// TIA Portal V20 export
FUNCTION_BLOCK "Sequence_1_JROutPnPLeft"   // FB32846, LAD
TITLE = Sequence
// Sequence template programmend in ladder logic
// stored: IsIECCheckEnabled true, MemoryReserve 100, Namespace Unit1.Em2, SetENOAutomatically true
   VAR_INPUT
      unitStatus : "LAF_typeUnitStatus";
   END_VAR
   VAR
      instSequenceLADControl { ExternalWritable := 'False'} : "LAF_ControlLadSequence";
      instSequenceLADStatus { ExternalWritable := 'False'} : "LAF_StatusLadSequence";
      statTonTime { ExternalWritable := 'False'} : Array[0..9999] of TON_TIME;
      NoDataCheck { S7_SetPoint := 'True'} : "LER_typePartData";
   END_VAR
   VAR_TEMP
      tempCustomerAction : Bool;   // Placeholder for possible actions
      tempDo_nothing_and_wait_for_init : Bool;   // Placeholder for doing nothing
      tempSafeStateCondition : Bool;   // Temp Condition for the equipment module to be in a safe state
   END_VAR
   VAR CONSTANT
      delayTime : Time := T#100ms;
      STEP_IDLE : DInt := 1;
      JOB_1_STEP_01 : DInt := 101;
      JOB_1_STEP_10 : DInt := 110;
      JOB_1_STEP_20 : DInt := 120;
      JOB_1_STEP_30 : DInt := 130;
      JOB_1_STEP_40 : DInt := 140;
      JOB_1_STEP_50 : DInt := 150;
      JOB_1_STEP_60 : DInt := 160;
      JOB_1_STEP_70 : DInt := 170;
      JOB_1_STEP_80 : DInt := 180;
      JOB_1_STEP_90 : DInt := 190;
      JOB_2_STEP_01 : DInt := 201;
      JOB_2_STEP_10 : DInt := 210;
      JOB_2_STEP_11 : DInt := 211;
      JOB_2_STEP_12 : DInt := 212;
      JOB_2_STEP_20 : DInt := 220;
      JOB_2_STEP_21 : DInt := 221;
      JOB_2_STEP_22 : DInt := 222;
      JOB_2_STEP_23 : DInt := 223;
      JOB_2_STEP_30 : DInt := 230;
      JOB_2_STEP_31 : DInt := 231;
      JOB_2_STEP_32 : DInt := 232;
      JOB_2_STEP_33 : DInt := 233;
      JOB_2_STEP_34 : DInt := 234;
      JOB_2_STEP_40 : DInt := 240;
      JOB_2_STEP_41 : DInt := 241;
      JOB_2_STEP_42 : DInt := 242;
      JOB_2_STEP_50 : DInt := 250;
      JOB_2_STEP_60 : DInt := 260;
      JOB_2_STEP_70 : DInt := 270;
      JOB_2_STEP_71 : DInt := 271;
      JOB_2_STEP_72 : DInt := 272;
      JOB_2_STEP_73 : DInt := 273;
      JOB_2_STEP_80 : DInt := 280;
      JOB_2_STEP_90 : DInt := 290;
      JOB_3_STEP_01 : DInt := 301;
      JOB_3_STEP_10 : DInt := 310;
      JOB_3_STEP_11 : DInt := 311;
      JOB_3_STEP_12 : DInt := 312;
      JOB_3_STEP_20 : DInt := 320;
      JOB_3_STEP_21 : DInt := 321;
      JOB_3_STEP_22 : DInt := 322;
      JOB_3_STEP_23 : DInt := 323;
      JOB_3_STEP_30 : DInt := 330;
      JOB_3_STEP_31 : DInt := 331;
      JOB_3_STEP_32 : DInt := 332;
      JOB_3_STEP_33 : DInt := 333;
      JOB_3_STEP_34 : DInt := 334;
      JOB_3_STEP_40 : DInt := 340;
      JOB_3_STEP_41 : DInt := 341;
      JOB_3_STEP_42 : DInt := 342;
      JOB_3_STEP_50 : DInt := 350;
      JOB_3_STEP_60 : DInt := 360;
      JOB_3_STEP_70 : DInt := 370;
      JOB_3_STEP_71 : DInt := 371;
      JOB_3_STEP_72 : DInt := 372;
      JOB_3_STEP_80 : DInt := 380;
      JOB_3_STEP_90 : DInt := 390;
      JOB_4_STEP_01 : DInt := 401;
      JOB_4_STEP_10 : DInt := 410;
      JOB_4_STEP_11 : DInt := 411;
      JOB_4_STEP_12 : DInt := 412;
      JOB_4_STEP_20 : DInt := 420;
      JOB_4_STEP_21 : DInt := 421;
      JOB_4_STEP_22 : DInt := 422;
      JOB_4_STEP_30 : DInt := 430;
      JOB_4_STEP_31 : DInt := 431;
      JOB_4_STEP_32 : DInt := 432;
      JOB_4_STEP_40 : DInt := 440;
      JOB_4_STEP_41 : DInt := 441;
      JOB_4_STEP_42 : DInt := 442;
      JOB_4_STEP_50 : DInt := 450;
      JOB_4_STEP_51 : DInt := 451;
      JOB_4_STEP_52 : DInt := 452;
      JOB_4_STEP_60 : DInt := 460;
      JOB_4_STEP_70 : DInt := 470;
      JOB_4_STEP_80 : DInt := 480;
      JOB_4_STEP_90 : DInt := 490;
      STEP_IMMEDIATE_STOP : DInt := 9001;   // Step executed when an immediate stop command is triggered for the sequence (i.e. when unit is in state aborting)
      TRUE : Bool := TRUE;
      FALSE : Bool := FALSE;
   END_VAR
   VAR_TEMP   // added for the SCL form of the ladder/FBD networks
      _w1 : Bool;
      _w2 : Bool;
      _w3 : Bool;
      _w4 : Bool;
      _w5 : Bool;
      _w6 : Bool;
      _w7 : Bool;
   END_VAR
BEGIN

REGION Network 1: BLOCK INFO HEADER
   // (company) / (C) Copyright (year)
   // ---------------------------------------------------------------------------------
   // Title:                             (Title of this block)
   // Comment/Function: (that is implemented in the block)
   // Library/Family:           (that the source is dedicated to)
   // Author:                        (department / person in charge / contact)
   // Target System:          (test system with FW version)
   // Engineering:              TIA Portal (SW version)
   // Restrictions:               (OB types, etc.)
   // Requirements:           (hardware, technological package, etc.)
   // ---------------------------------------------------------------------------------
   // Change log table:
   // Version          | Date             | Signature      | Expert in charge  | Changes applied ------------------------|----------------------|-------------------------|--------------------------------|-----------------------
   // 001.000.000 | yyyy-mm-dd | 0x00000000 | (name of expert) | First released version
END_REGION

REGION Network 2: DESCRIPTION
   // This is a template block provided by the Automation Framework. It can be used to create an own project.
   // The Block Info Header is prepared to put in your own data.
   // Description of the block could be added here and the docu created by Code2Docu.
END_REGION

REGION Network 3: *************** CONTROL **********************
END_REGION

REGION Network 4: Sequence Control ("Enter your Sequins number here")
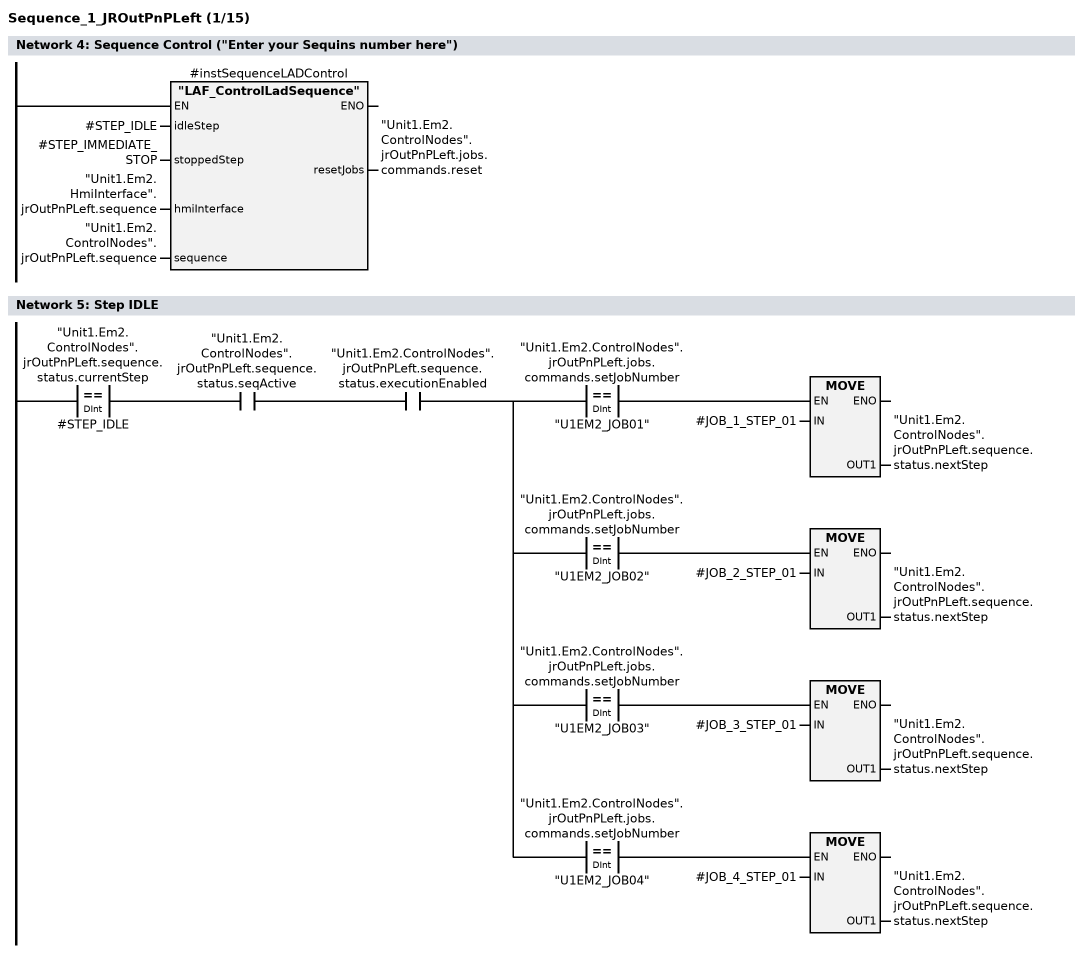
   RUNG wire#powerrail
      #instSequenceLADControl(idleStep := #STEP_IDLE, stoppedStep := #STEP_IMMEDIATE_STOP, hmiInterface := "Unit1.Em2.HmiInterface".jrOutPnPLeft.sequence, sequence := "Unit1.Em2.ControlNodes".jrOutPnPLeft.sequence, resetJobs => "Unit1.Em2.ControlNodes".jrOutPnPLeft.jobs.commands.reset)
   END_RUNG
   // the same network as SCL:
   #instSequenceLADControl(idleStep := #STEP_IDLE,   // "LAF_ControlLadSequence"
                           stoppedStep := #STEP_IMMEDIATE_STOP,
                           hmiInterface := "Unit1.Em2.HmiInterface".jrOutPnPLeft.sequence,
                           sequence := "Unit1.Em2.ControlNodes".jrOutPnPLeft.sequence,
                           resetJobs => "Unit1.Em2.ControlNodes".jrOutPnPLeft.jobs.commands.reset);
END_REGION

REGION Network 5: Step IDLE
   RUNG wire#powerrail
      { S7_Templates := "SrcType := DInt" } EQ_Contact(in1 := "Unit1.Em2.ControlNodes".jrOutPnPLeft.sequence.status.currentStep, in2 := #STEP_IDLE)
      Contact( "Unit1.Em2.ControlNodes".jrOutPnPLeft.sequence.status.seqActive )
      Contact( "Unit1.Em2.ControlNodes".jrOutPnPLeft.sequence.status.executionEnabled )
      wire#w1
      { S7_Templates := "SrcType := DInt" } EQ_Contact(in1 := "Unit1.Em2.ControlNodes".jrOutPnPLeft.jobs.commands.setJobNumber, in2 := "U1EM2_JOB01")
      Move(in := #JOB_1_STEP_01, out1 => "Unit1.Em2.ControlNodes".jrOutPnPLeft.sequence.status.nextStep)
   END_RUNG
   RUNG wire#w1
      { S7_Templates := "SrcType := DInt" } EQ_Contact(in1 := "Unit1.Em2.ControlNodes".jrOutPnPLeft.jobs.commands.setJobNumber, in2 := "U1EM2_JOB02")
      Move(in := #JOB_2_STEP_01, out1 => "Unit1.Em2.ControlNodes".jrOutPnPLeft.sequence.status.nextStep)
   END_RUNG
   RUNG wire#w1
      { S7_Templates := "SrcType := DInt" } EQ_Contact(in1 := "Unit1.Em2.ControlNodes".jrOutPnPLeft.jobs.commands.setJobNumber, in2 := "U1EM2_JOB03")
      Move(in := #JOB_3_STEP_01, out1 => "Unit1.Em2.ControlNodes".jrOutPnPLeft.sequence.status.nextStep)
   END_RUNG
   RUNG wire#w1
      { S7_Templates := "SrcType := DInt" } EQ_Contact(in1 := "Unit1.Em2.ControlNodes".jrOutPnPLeft.jobs.commands.setJobNumber, in2 := "U1EM2_JOB04")
      Move(in := #JOB_4_STEP_01, out1 => "Unit1.Em2.ControlNodes".jrOutPnPLeft.sequence.status.nextStep)
   END_RUNG
   // the same network as SCL:
   #_w1 := ("Unit1.Em2.ControlNodes".jrOutPnPLeft.sequence.status.currentStep = #STEP_IDLE) AND "Unit1.Em2.ControlNodes".jrOutPnPLeft.sequence.status.seqActive AND "Unit1.Em2.ControlNodes".jrOutPnPLeft.sequence.status.executionEnabled;
   IF #_w1 AND ("Unit1.Em2.ControlNodes".jrOutPnPLeft.jobs.commands.setJobNumber = "U1EM2_JOB01") THEN
       "Unit1.Em2.ControlNodes".jrOutPnPLeft.sequence.status.nextStep := #JOB_1_STEP_01;
   END_IF;
   IF #_w1 AND ("Unit1.Em2.ControlNodes".jrOutPnPLeft.jobs.commands.setJobNumber = "U1EM2_JOB02") THEN
       "Unit1.Em2.ControlNodes".jrOutPnPLeft.sequence.status.nextStep := #JOB_2_STEP_01;
   END_IF;
   IF #_w1 AND ("Unit1.Em2.ControlNodes".jrOutPnPLeft.jobs.commands.setJobNumber = "U1EM2_JOB03") THEN
       "Unit1.Em2.ControlNodes".jrOutPnPLeft.sequence.status.nextStep := #JOB_3_STEP_01;
   END_IF;
   IF #_w1 AND ("Unit1.Em2.ControlNodes".jrOutPnPLeft.jobs.commands.setJobNumber = "U1EM2_JOB04") THEN
       "Unit1.Em2.ControlNodes".jrOutPnPLeft.sequence.status.nextStep := #JOB_4_STEP_01;
   END_IF;
END_REGION

REGION Network 6: *************** JOB[1] EM HOMING *************************
END_REGION

REGION Network 7: Step[101] : JOB[1] Condition
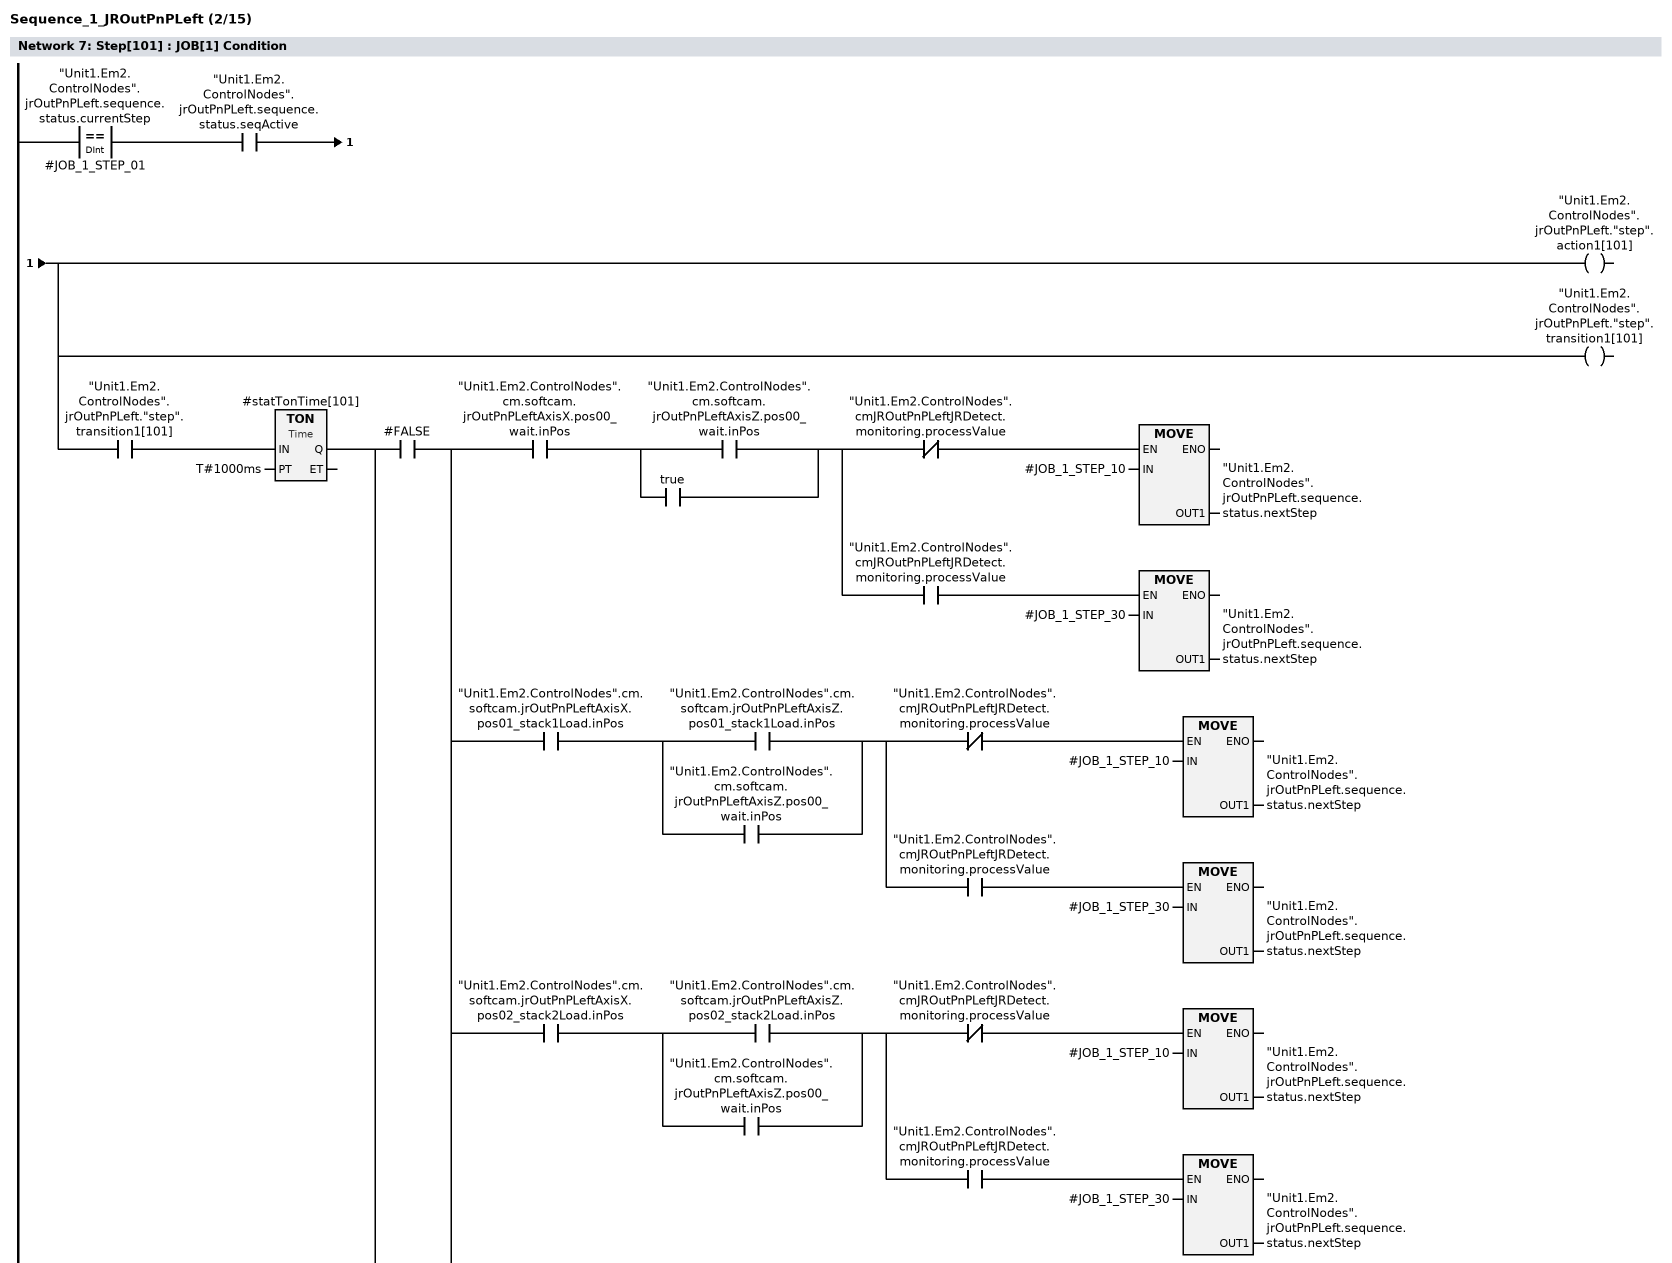
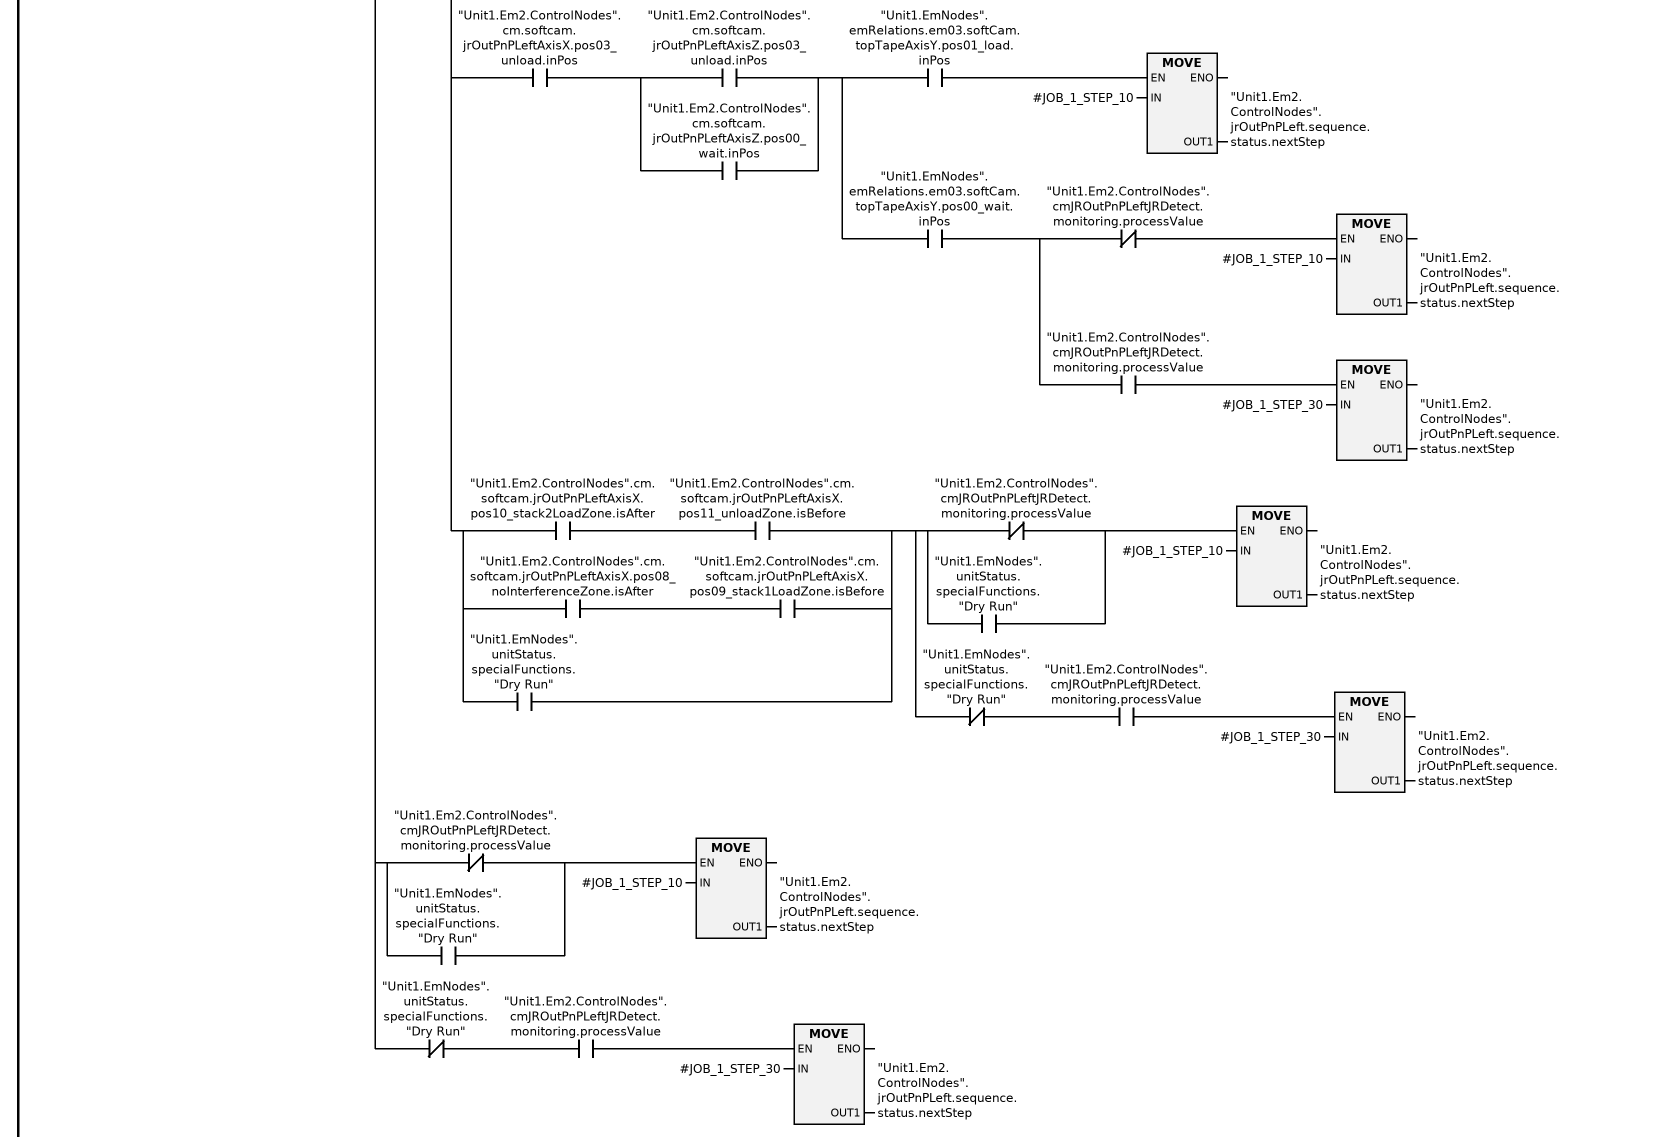
   RUNG wire#powerrail
      { S7_Templates := "SrcType := DInt" } EQ_Contact(in1 := "Unit1.Em2.ControlNodes".jrOutPnPLeft.sequence.status.currentStep, in2 := #JOB_1_STEP_01)
      Contact( "Unit1.Em2.ControlNodes".jrOutPnPLeft.sequence.status.seqActive )
      wire#w1
      Coil( "Unit1.Em2.ControlNodes".jrOutPnPLeft."step".action1[101] )
   END_RUNG
   RUNG wire#w1
      Coil( "Unit1.Em2.ControlNodes".jrOutPnPLeft."step".transition1[101] )
   END_RUNG
   RUNG wire#w1
      Contact( "Unit1.Em2.ControlNodes".jrOutPnPLeft."step".transition1[101] )
      { S7_Templates := "time_type := Time" } #statTonTime[101].TON(pt := T#1000ms, et =>)
      wire#w2
      Contact( #FALSE )
      wire#w3
      Contact( "Unit1.Em2.ControlNodes".cm.softcam.jrOutPnPLeftAxisX.pos00_wait.inPos )
      wire#w4
      Contact( "Unit1.Em2.ControlNodes".cm.softcam.jrOutPnPLeftAxisZ.pos00_wait.inPos )
      wire#w5
      I_Contact( "Unit1.Em2.ControlNodes".cmJROutPnPLeftJRDetect.monitoring.processValue )
      Move(in := #JOB_1_STEP_10, out1 => "Unit1.Em2.ControlNodes".jrOutPnPLeft.sequence.status.nextStep)
   END_RUNG
   RUNG wire#w4
      Contact( true )
   END_RUNG wire#w5
   RUNG wire#w5
      Contact( "Unit1.Em2.ControlNodes".cmJROutPnPLeftJRDetect.monitoring.processValue )
      Move(in := #JOB_1_STEP_30, out1 => "Unit1.Em2.ControlNodes".jrOutPnPLeft.sequence.status.nextStep)
   END_RUNG
   RUNG wire#w3
      Contact( "Unit1.Em2.ControlNodes".cm.softcam.jrOutPnPLeftAxisX.pos01_stack1Load.inPos )
      wire#w6
      Contact( "Unit1.Em2.ControlNodes".cm.softcam.jrOutPnPLeftAxisZ.pos01_stack1Load.inPos )
      wire#w7
      I_Contact( "Unit1.Em2.ControlNodes".cmJROutPnPLeftJRDetect.monitoring.processValue )
      Move(in := #JOB_1_STEP_10, out1 => "Unit1.Em2.ControlNodes".jrOutPnPLeft.sequence.status.nextStep)
   END_RUNG
   RUNG wire#w6
      Contact( "Unit1.Em2.ControlNodes".cm.softcam.jrOutPnPLeftAxisZ.pos00_wait.inPos )
   END_RUNG wire#w7
   RUNG wire#w7
      Contact( "Unit1.Em2.ControlNodes".cmJROutPnPLeftJRDetect.monitoring.processValue )
      Move(in := #JOB_1_STEP_30, out1 => "Unit1.Em2.ControlNodes".jrOutPnPLeft.sequence.status.nextStep)
   END_RUNG
   RUNG wire#w3
      Contact( "Unit1.Em2.ControlNodes".cm.softcam.jrOutPnPLeftAxisX.pos02_stack2Load.inPos )
      wire#w8
      Contact( "Unit1.Em2.ControlNodes".cm.softcam.jrOutPnPLeftAxisZ.pos02_stack2Load.inPos )
      wire#w9
      I_Contact( "Unit1.Em2.ControlNodes".cmJROutPnPLeftJRDetect.monitoring.processValue )
      Move(in := #JOB_1_STEP_10, out1 => "Unit1.Em2.ControlNodes".jrOutPnPLeft.sequence.status.nextStep)
   END_RUNG
   RUNG wire#w8
      Contact( "Unit1.Em2.ControlNodes".cm.softcam.jrOutPnPLeftAxisZ.pos00_wait.inPos )
   END_RUNG wire#w9
   RUNG wire#w9
      Contact( "Unit1.Em2.ControlNodes".cmJROutPnPLeftJRDetect.monitoring.processValue )
      Move(in := #JOB_1_STEP_30, out1 => "Unit1.Em2.ControlNodes".jrOutPnPLeft.sequence.status.nextStep)
   END_RUNG
   RUNG wire#w3
      Contact( "Unit1.Em2.ControlNodes".cm.softcam.jrOutPnPLeftAxisX.pos03_unload.inPos )
      wire#w10
      Contact( "Unit1.Em2.ControlNodes".cm.softcam.jrOutPnPLeftAxisZ.pos03_unload.inPos )
      wire#w11
      Contact( "Unit1.EmNodes".emRelations.em03.softCam.topTapeAxisY.pos01_load.inPos )
      Move(in := #JOB_1_STEP_10, out1 => "Unit1.Em2.ControlNodes".jrOutPnPLeft.sequence.status.nextStep)
   END_RUNG
   RUNG wire#w10
      Contact( "Unit1.Em2.ControlNodes".cm.softcam.jrOutPnPLeftAxisZ.pos00_wait.inPos )
   END_RUNG wire#w11
   RUNG wire#w11
      Contact( "Unit1.EmNodes".emRelations.em03.softCam.topTapeAxisY.pos00_wait.inPos )
      wire#w12
      I_Contact( "Unit1.Em2.ControlNodes".cmJROutPnPLeftJRDetect.monitoring.processValue )
      Move(in := #JOB_1_STEP_10, out1 => "Unit1.Em2.ControlNodes".jrOutPnPLeft.sequence.status.nextStep)
   END_RUNG
   RUNG wire#w12
      Contact( "Unit1.Em2.ControlNodes".cmJROutPnPLeftJRDetect.monitoring.processValue )
      Move(in := #JOB_1_STEP_30, out1 => "Unit1.Em2.ControlNodes".jrOutPnPLeft.sequence.status.nextStep)
   END_RUNG
   RUNG wire#w3
      Contact( "Unit1.Em2.ControlNodes".cm.softcam.jrOutPnPLeftAxisX.pos10_stack2LoadZone.isAfter )
      Contact( "Unit1.Em2.ControlNodes".cm.softcam.jrOutPnPLeftAxisX.pos11_unloadZone.isBefore )
      wire#w13
      I_Contact( "Unit1.Em2.ControlNodes".cmJROutPnPLeftJRDetect.monitoring.processValue )
      wire#w14
      Move(in := #JOB_1_STEP_10, out1 => "Unit1.Em2.ControlNodes".jrOutPnPLeft.sequence.status.nextStep)
   END_RUNG
   RUNG wire#w3
      Contact( "Unit1.Em2.ControlNodes".cm.softcam.jrOutPnPLeftAxisX.pos08_noInterferenceZone.isAfter )
      Contact( "Unit1.Em2.ControlNodes".cm.softcam.jrOutPnPLeftAxisX.pos09_stack1LoadZone.isBefore )
   END_RUNG wire#w13
   RUNG wire#w3
      Contact( "Unit1.EmNodes".unitStatus.specialFunctions."Dry Run" )
   END_RUNG wire#w13
   RUNG wire#w13
      Contact( "Unit1.EmNodes".unitStatus.specialFunctions."Dry Run" )
   END_RUNG wire#w14
   RUNG wire#w13
      I_Contact( "Unit1.EmNodes".unitStatus.specialFunctions."Dry Run" )
      Contact( "Unit1.Em2.ControlNodes".cmJROutPnPLeftJRDetect.monitoring.processValue )
      Move(in := #JOB_1_STEP_30, out1 => "Unit1.Em2.ControlNodes".jrOutPnPLeft.sequence.status.nextStep)
   END_RUNG
   RUNG wire#w2
      I_Contact( "Unit1.Em2.ControlNodes".cmJROutPnPLeftJRDetect.monitoring.processValue )
      wire#w15
      Move(in := #JOB_1_STEP_10, out1 => "Unit1.Em2.ControlNodes".jrOutPnPLeft.sequence.status.nextStep)
   END_RUNG
   RUNG wire#w2
      Contact( "Unit1.EmNodes".unitStatus.specialFunctions."Dry Run" )
   END_RUNG wire#w15
   RUNG wire#w2
      I_Contact( "Unit1.EmNodes".unitStatus.specialFunctions."Dry Run" )
      Contact( "Unit1.Em2.ControlNodes".cmJROutPnPLeftJRDetect.monitoring.processValue )
      Move(in := #JOB_1_STEP_30, out1 => "Unit1.Em2.ControlNodes".jrOutPnPLeft.sequence.status.nextStep)
   END_RUNG
   // the same network as SCL:
   "Unit1.Em2.ControlNodes".jrOutPnPLeft."step".action1[101] := ("Unit1.Em2.ControlNodes".jrOutPnPLeft.sequence.status.currentStep = #JOB_1_STEP_01) AND "Unit1.Em2.ControlNodes".jrOutPnPLeft.sequence.status.seqActive;
   "Unit1.Em2.ControlNodes".jrOutPnPLeft."step".transition1[101] := ("Unit1.Em2.ControlNodes".jrOutPnPLeft.sequence.status.currentStep = #JOB_1_STEP_01) AND "Unit1.Em2.ControlNodes".jrOutPnPLeft.sequence.status.seqActive;
   #statTonTime[101].TON(IN := ("Unit1.Em2.ControlNodes".jrOutPnPLeft.sequence.status.currentStep = #JOB_1_STEP_01) AND "Unit1.Em2.ControlNodes".jrOutPnPLeft.sequence.status.seqActive AND "Unit1.Em2.ControlNodes".jrOutPnPLeft."step".transition1[101],
                         PT := T#1000ms);
   #_w1 := #statTonTime[101].Q AND #FALSE;
   #_w2 := #_w1 AND "Unit1.Em2.ControlNodes".cm.softcam.jrOutPnPLeftAxisX.pos00_wait.inPos AND ("Unit1.Em2.ControlNodes".cm.softcam.jrOutPnPLeftAxisZ.pos00_wait.inPos OR true);
   IF #_w2 AND NOT "Unit1.Em2.ControlNodes".cmJROutPnPLeftJRDetect.monitoring.processValue THEN
       "Unit1.Em2.ControlNodes".jrOutPnPLeft.sequence.status.nextStep := #JOB_1_STEP_10;
   END_IF;
   IF #_w2 AND "Unit1.Em2.ControlNodes".cmJROutPnPLeftJRDetect.monitoring.processValue THEN
       "Unit1.Em2.ControlNodes".jrOutPnPLeft.sequence.status.nextStep := #JOB_1_STEP_30;
   END_IF;
   #_w3 := #_w1 AND "Unit1.Em2.ControlNodes".cm.softcam.jrOutPnPLeftAxisX.pos01_stack1Load.inPos AND ("Unit1.Em2.ControlNodes".cm.softcam.jrOutPnPLeftAxisZ.pos01_stack1Load.inPos OR "Unit1.Em2.ControlNodes".cm.softcam.jrOutPnPLeftAxisZ.pos00_wait.inPos);
   IF #_w3 AND NOT "Unit1.Em2.ControlNodes".cmJROutPnPLeftJRDetect.monitoring.processValue THEN
       "Unit1.Em2.ControlNodes".jrOutPnPLeft.sequence.status.nextStep := #JOB_1_STEP_10;
   END_IF;
   IF #_w3 AND "Unit1.Em2.ControlNodes".cmJROutPnPLeftJRDetect.monitoring.processValue THEN
       "Unit1.Em2.ControlNodes".jrOutPnPLeft.sequence.status.nextStep := #JOB_1_STEP_30;
   END_IF;
   #_w4 := #_w1 AND "Unit1.Em2.ControlNodes".cm.softcam.jrOutPnPLeftAxisX.pos02_stack2Load.inPos AND ("Unit1.Em2.ControlNodes".cm.softcam.jrOutPnPLeftAxisZ.pos02_stack2Load.inPos OR "Unit1.Em2.ControlNodes".cm.softcam.jrOutPnPLeftAxisZ.pos00_wait.inPos);
   IF #_w4 AND NOT "Unit1.Em2.ControlNodes".cmJROutPnPLeftJRDetect.monitoring.processValue THEN
       "Unit1.Em2.ControlNodes".jrOutPnPLeft.sequence.status.nextStep := #JOB_1_STEP_10;
   END_IF;
   IF #_w4 AND "Unit1.Em2.ControlNodes".cmJROutPnPLeftJRDetect.monitoring.processValue THEN
       "Unit1.Em2.ControlNodes".jrOutPnPLeft.sequence.status.nextStep := #JOB_1_STEP_30;
   END_IF;
   #_w5 := #_w1 AND "Unit1.Em2.ControlNodes".cm.softcam.jrOutPnPLeftAxisX.pos03_unload.inPos AND ("Unit1.Em2.ControlNodes".cm.softcam.jrOutPnPLeftAxisZ.pos03_unload.inPos OR "Unit1.Em2.ControlNodes".cm.softcam.jrOutPnPLeftAxisZ.pos00_wait.inPos);
   IF #_w5 AND "Unit1.EmNodes".emRelations.em03.softCam.topTapeAxisY.pos01_load.inPos THEN
       "Unit1.Em2.ControlNodes".jrOutPnPLeft.sequence.status.nextStep := #JOB_1_STEP_10;
   END_IF;
   #_w6 := #_w5 AND "Unit1.EmNodes".emRelations.em03.softCam.topTapeAxisY.pos00_wait.inPos;
   IF #_w6 AND NOT "Unit1.Em2.ControlNodes".cmJROutPnPLeftJRDetect.monitoring.processValue THEN
       "Unit1.Em2.ControlNodes".jrOutPnPLeft.sequence.status.nextStep := #JOB_1_STEP_10;
   END_IF;
   IF #_w6 AND "Unit1.Em2.ControlNodes".cmJROutPnPLeftJRDetect.monitoring.processValue THEN
       "Unit1.Em2.ControlNodes".jrOutPnPLeft.sequence.status.nextStep := #JOB_1_STEP_30;
   END_IF;
   #_w7 := #_w1 AND (("Unit1.Em2.ControlNodes".cm.softcam.jrOutPnPLeftAxisX.pos10_stack2LoadZone.isAfter AND "Unit1.Em2.ControlNodes".cm.softcam.jrOutPnPLeftAxisX.pos11_unloadZone.isBefore) OR ("Unit1.Em2.ControlNodes".cm.softcam.jrOutPnPLeftAxisX.pos08_noInterferenceZone.isAfter AND "Unit1.Em2.ControlNodes".cm.softcam.jrOutPnPLeftAxisX.pos09_stack1LoadZone.isBefore) OR "Unit1.EmNodes".unitStatus.specialFunctions."Dry Run");
   IF #_w7 AND (NOT "Unit1.Em2.ControlNodes".cmJROutPnPLeftJRDetect.monitoring.processValue OR "Unit1.EmNodes".unitStatus.specialFunctions."Dry Run") THEN
       "Unit1.Em2.ControlNodes".jrOutPnPLeft.sequence.status.nextStep := #JOB_1_STEP_10;
   END_IF;
   IF #_w7 AND NOT "Unit1.EmNodes".unitStatus.specialFunctions."Dry Run" AND "Unit1.Em2.ControlNodes".cmJROutPnPLeftJRDetect.monitoring.processValue THEN
       "Unit1.Em2.ControlNodes".jrOutPnPLeft.sequence.status.nextStep := #JOB_1_STEP_30;
   END_IF;
   IF #statTonTime[101].Q AND (NOT "Unit1.Em2.ControlNodes".cmJROutPnPLeftJRDetect.monitoring.processValue OR "Unit1.EmNodes".unitStatus.specialFunctions."Dry Run") THEN
       "Unit1.Em2.ControlNodes".jrOutPnPLeft.sequence.status.nextStep := #JOB_1_STEP_10;
   END_IF;
   IF #statTonTime[101].Q AND NOT "Unit1.EmNodes".unitStatus.specialFunctions."Dry Run" AND "Unit1.Em2.ControlNodes".cmJROutPnPLeftJRDetect.monitoring.processValue THEN
       "Unit1.Em2.ControlNodes".jrOutPnPLeft.sequence.status.nextStep := #JOB_1_STEP_30;
   END_IF;
END_REGION

REGION Network 8: Step[110] : JR PP Left Clamp Open
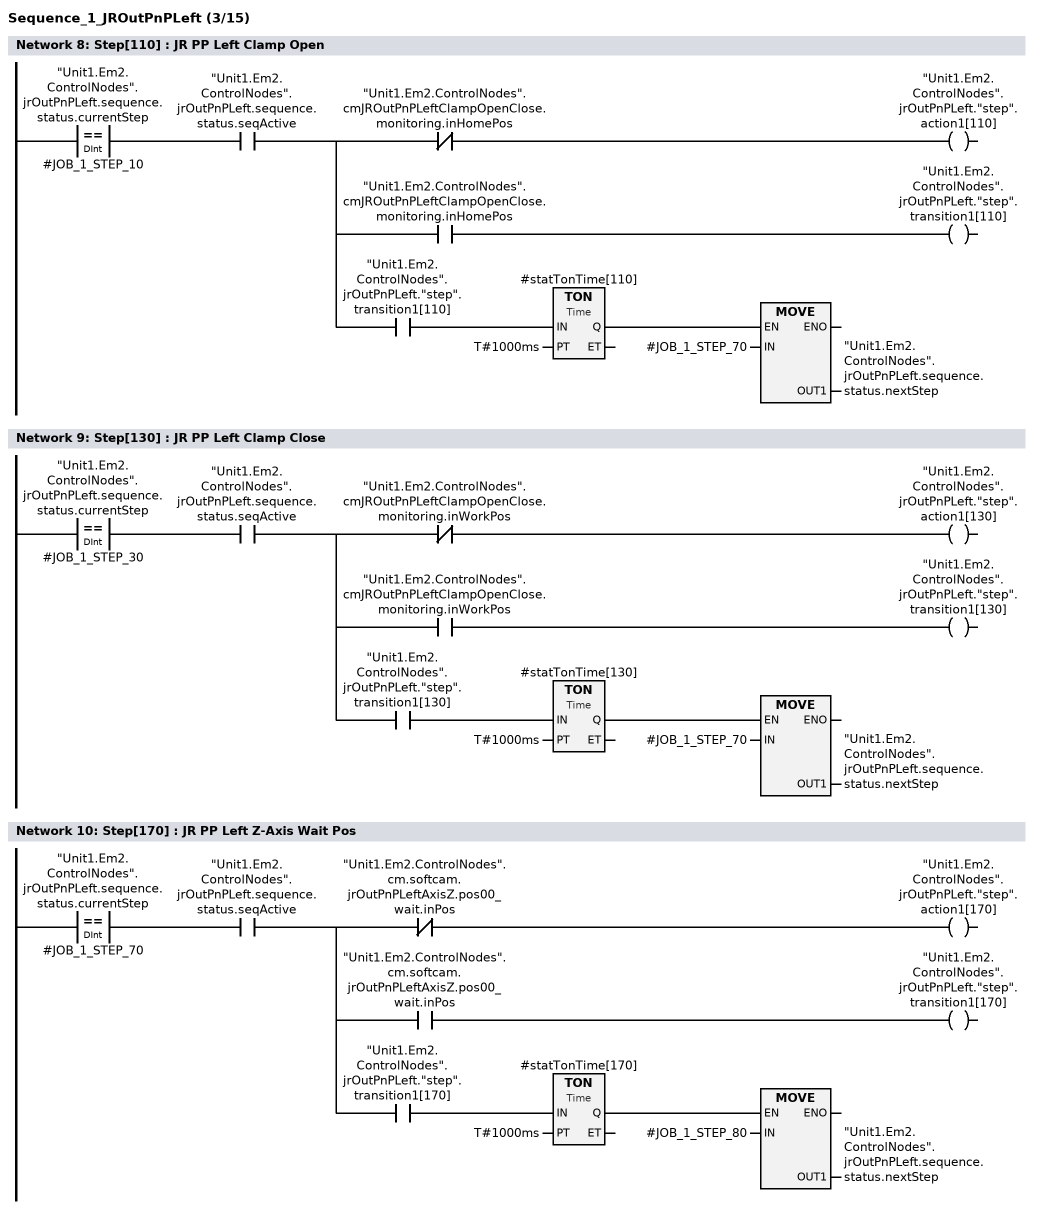
   RUNG wire#powerrail
      { S7_Templates := "SrcType := DInt" } EQ_Contact(in1 := "Unit1.Em2.ControlNodes".jrOutPnPLeft.sequence.status.currentStep, in2 := #JOB_1_STEP_10)
      Contact( "Unit1.Em2.ControlNodes".jrOutPnPLeft.sequence.status.seqActive )
      wire#w1
      I_Contact( "Unit1.Em2.ControlNodes".cmJROutPnPLeftClampOpenClose.monitoring.inHomePos )
      Coil( "Unit1.Em2.ControlNodes".jrOutPnPLeft."step".action1[110] )
   END_RUNG
   RUNG wire#w1
      Contact( "Unit1.Em2.ControlNodes".cmJROutPnPLeftClampOpenClose.monitoring.inHomePos )
      Coil( "Unit1.Em2.ControlNodes".jrOutPnPLeft."step".transition1[110] )
   END_RUNG
   RUNG wire#w1
      Contact( "Unit1.Em2.ControlNodes".jrOutPnPLeft."step".transition1[110] )
      { S7_Templates := "time_type := Time" } #statTonTime[110].TON(pt := T#1000ms, et =>)
      Move(in := #JOB_1_STEP_70, out1 => "Unit1.Em2.ControlNodes".jrOutPnPLeft.sequence.status.nextStep)
   END_RUNG
   // the same network as SCL:
   #_w1 := ("Unit1.Em2.ControlNodes".jrOutPnPLeft.sequence.status.currentStep = #JOB_1_STEP_10) AND "Unit1.Em2.ControlNodes".jrOutPnPLeft.sequence.status.seqActive;
   "Unit1.Em2.ControlNodes".jrOutPnPLeft."step".action1[110] := #_w1 AND NOT "Unit1.Em2.ControlNodes".cmJROutPnPLeftClampOpenClose.monitoring.inHomePos;
   "Unit1.Em2.ControlNodes".jrOutPnPLeft."step".transition1[110] := #_w1 AND "Unit1.Em2.ControlNodes".cmJROutPnPLeftClampOpenClose.monitoring.inHomePos;
   #statTonTime[110].TON(IN := #_w1 AND "Unit1.Em2.ControlNodes".jrOutPnPLeft."step".transition1[110],
                         PT := T#1000ms);
   IF #statTonTime[110].Q THEN
       "Unit1.Em2.ControlNodes".jrOutPnPLeft.sequence.status.nextStep := #JOB_1_STEP_70;
   END_IF;
END_REGION

REGION Network 9: Step[130] : JR PP Left Clamp Close
   RUNG wire#powerrail
      { S7_Templates := "SrcType := DInt" } EQ_Contact(in1 := "Unit1.Em2.ControlNodes".jrOutPnPLeft.sequence.status.currentStep, in2 := #JOB_1_STEP_30)
      Contact( "Unit1.Em2.ControlNodes".jrOutPnPLeft.sequence.status.seqActive )
      wire#w1
      I_Contact( "Unit1.Em2.ControlNodes".cmJROutPnPLeftClampOpenClose.monitoring.inWorkPos )
      Coil( "Unit1.Em2.ControlNodes".jrOutPnPLeft."step".action1[130] )
   END_RUNG
   RUNG wire#w1
      Contact( "Unit1.Em2.ControlNodes".cmJROutPnPLeftClampOpenClose.monitoring.inWorkPos )
      Coil( "Unit1.Em2.ControlNodes".jrOutPnPLeft."step".transition1[130] )
   END_RUNG
   RUNG wire#w1
      Contact( "Unit1.Em2.ControlNodes".jrOutPnPLeft."step".transition1[130] )
      { S7_Templates := "time_type := Time" } #statTonTime[130].TON(pt := T#1000ms, et =>)
      Move(in := #JOB_1_STEP_70, out1 => "Unit1.Em2.ControlNodes".jrOutPnPLeft.sequence.status.nextStep)
   END_RUNG
   // the same network as SCL:
   #_w1 := ("Unit1.Em2.ControlNodes".jrOutPnPLeft.sequence.status.currentStep = #JOB_1_STEP_30) AND "Unit1.Em2.ControlNodes".jrOutPnPLeft.sequence.status.seqActive;
   "Unit1.Em2.ControlNodes".jrOutPnPLeft."step".action1[130] := #_w1 AND NOT "Unit1.Em2.ControlNodes".cmJROutPnPLeftClampOpenClose.monitoring.inWorkPos;
   "Unit1.Em2.ControlNodes".jrOutPnPLeft."step".transition1[130] := #_w1 AND "Unit1.Em2.ControlNodes".cmJROutPnPLeftClampOpenClose.monitoring.inWorkPos;
   #statTonTime[130].TON(IN := #_w1 AND "Unit1.Em2.ControlNodes".jrOutPnPLeft."step".transition1[130],
                         PT := T#1000ms);
   IF #statTonTime[130].Q THEN
       "Unit1.Em2.ControlNodes".jrOutPnPLeft.sequence.status.nextStep := #JOB_1_STEP_70;
   END_IF;
END_REGION

REGION Network 10: Step[170] : JR PP Left Z-Axis Wait Pos
   RUNG wire#powerrail
      { S7_Templates := "SrcType := DInt" } EQ_Contact(in1 := "Unit1.Em2.ControlNodes".jrOutPnPLeft.sequence.status.currentStep, in2 := #JOB_1_STEP_70)
      Contact( "Unit1.Em2.ControlNodes".jrOutPnPLeft.sequence.status.seqActive )
      wire#w1
      I_Contact( "Unit1.Em2.ControlNodes".cm.softcam.jrOutPnPLeftAxisZ.pos00_wait.inPos )
      Coil( "Unit1.Em2.ControlNodes".jrOutPnPLeft."step".action1[170] )
   END_RUNG
   RUNG wire#w1
      Contact( "Unit1.Em2.ControlNodes".cm.softcam.jrOutPnPLeftAxisZ.pos00_wait.inPos )
      Coil( "Unit1.Em2.ControlNodes".jrOutPnPLeft."step".transition1[170] )
   END_RUNG
   RUNG wire#w1
      Contact( "Unit1.Em2.ControlNodes".jrOutPnPLeft."step".transition1[170] )
      { S7_Templates := "time_type := Time" } #statTonTime[170].TON(pt := T#1000ms, et =>)
      Move(in := #JOB_1_STEP_80, out1 => "Unit1.Em2.ControlNodes".jrOutPnPLeft.sequence.status.nextStep)
   END_RUNG
   // the same network as SCL:
   #_w1 := ("Unit1.Em2.ControlNodes".jrOutPnPLeft.sequence.status.currentStep = #JOB_1_STEP_70) AND "Unit1.Em2.ControlNodes".jrOutPnPLeft.sequence.status.seqActive;
   "Unit1.Em2.ControlNodes".jrOutPnPLeft."step".action1[170] := #_w1 AND NOT "Unit1.Em2.ControlNodes".cm.softcam.jrOutPnPLeftAxisZ.pos00_wait.inPos;
   "Unit1.Em2.ControlNodes".jrOutPnPLeft."step".transition1[170] := #_w1 AND "Unit1.Em2.ControlNodes".cm.softcam.jrOutPnPLeftAxisZ.pos00_wait.inPos;
   #statTonTime[170].TON(IN := #_w1 AND "Unit1.Em2.ControlNodes".jrOutPnPLeft."step".transition1[170],
                         PT := T#1000ms);
   IF #statTonTime[170].Q THEN
       "Unit1.Em2.ControlNodes".jrOutPnPLeft.sequence.status.nextStep := #JOB_1_STEP_80;
   END_IF;
END_REGION

REGION Network 11: Step[180] : JR PP Left X-Axis Wait Pos
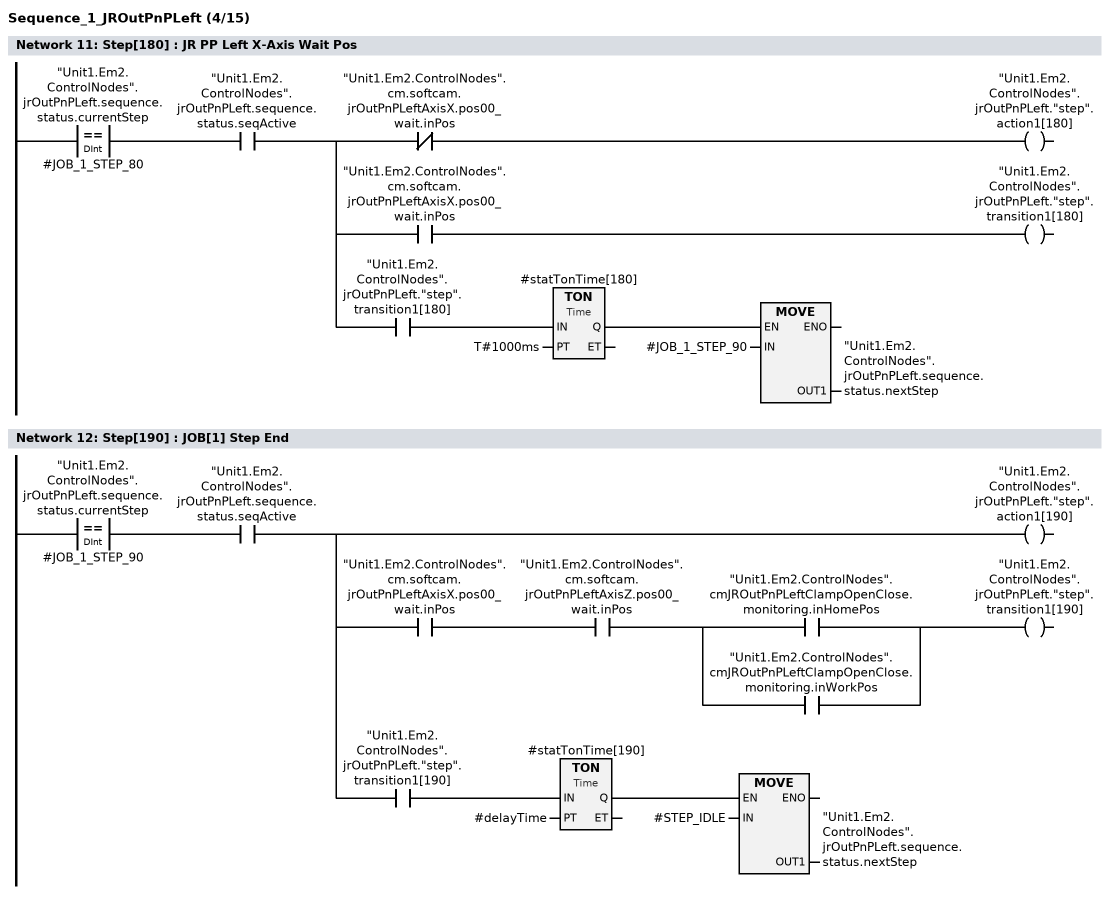
   RUNG wire#powerrail
      { S7_Templates := "SrcType := DInt" } EQ_Contact(in1 := "Unit1.Em2.ControlNodes".jrOutPnPLeft.sequence.status.currentStep, in2 := #JOB_1_STEP_80)
      Contact( "Unit1.Em2.ControlNodes".jrOutPnPLeft.sequence.status.seqActive )
      wire#w1
      I_Contact( "Unit1.Em2.ControlNodes".cm.softcam.jrOutPnPLeftAxisX.pos00_wait.inPos )
      Coil( "Unit1.Em2.ControlNodes".jrOutPnPLeft."step".action1[180] )
   END_RUNG
   RUNG wire#w1
      Contact( "Unit1.Em2.ControlNodes".cm.softcam.jrOutPnPLeftAxisX.pos00_wait.inPos )
      Coil( "Unit1.Em2.ControlNodes".jrOutPnPLeft."step".transition1[180] )
   END_RUNG
   RUNG wire#w1
      Contact( "Unit1.Em2.ControlNodes".jrOutPnPLeft."step".transition1[180] )
      { S7_Templates := "time_type := Time" } #statTonTime[180].TON(pt := T#1000ms, et =>)
      Move(in := #JOB_1_STEP_90, out1 => "Unit1.Em2.ControlNodes".jrOutPnPLeft.sequence.status.nextStep)
   END_RUNG
   // the same network as SCL:
   #_w1 := ("Unit1.Em2.ControlNodes".jrOutPnPLeft.sequence.status.currentStep = #JOB_1_STEP_80) AND "Unit1.Em2.ControlNodes".jrOutPnPLeft.sequence.status.seqActive;
   "Unit1.Em2.ControlNodes".jrOutPnPLeft."step".action1[180] := #_w1 AND NOT "Unit1.Em2.ControlNodes".cm.softcam.jrOutPnPLeftAxisX.pos00_wait.inPos;
   "Unit1.Em2.ControlNodes".jrOutPnPLeft."step".transition1[180] := #_w1 AND "Unit1.Em2.ControlNodes".cm.softcam.jrOutPnPLeftAxisX.pos00_wait.inPos;
   #statTonTime[180].TON(IN := #_w1 AND "Unit1.Em2.ControlNodes".jrOutPnPLeft."step".transition1[180],
                         PT := T#1000ms);
   IF #statTonTime[180].Q THEN
       "Unit1.Em2.ControlNodes".jrOutPnPLeft.sequence.status.nextStep := #JOB_1_STEP_90;
   END_IF;
END_REGION

REGION Network 12: Step[190] : JOB[1] Step End
   RUNG wire#powerrail
      { S7_Templates := "SrcType := DInt" } EQ_Contact(in1 := "Unit1.Em2.ControlNodes".jrOutPnPLeft.sequence.status.currentStep, in2 := #JOB_1_STEP_90)
      Contact( "Unit1.Em2.ControlNodes".jrOutPnPLeft.sequence.status.seqActive )
      wire#w1
      Coil( "Unit1.Em2.ControlNodes".jrOutPnPLeft."step".action1[190] )
   END_RUNG
   RUNG wire#w1
      Contact( "Unit1.Em2.ControlNodes".cm.softcam.jrOutPnPLeftAxisX.pos00_wait.inPos )
      Contact( "Unit1.Em2.ControlNodes".cm.softcam.jrOutPnPLeftAxisZ.pos00_wait.inPos )
      wire#w2
      Contact( "Unit1.Em2.ControlNodes".cmJROutPnPLeftClampOpenClose.monitoring.inHomePos )
      wire#w3
      Coil( "Unit1.Em2.ControlNodes".jrOutPnPLeft."step".transition1[190] )
   END_RUNG
   RUNG wire#w2
      Contact( "Unit1.Em2.ControlNodes".cmJROutPnPLeftClampOpenClose.monitoring.inWorkPos )
   END_RUNG wire#w3
   RUNG wire#w1
      Contact( "Unit1.Em2.ControlNodes".jrOutPnPLeft."step".transition1[190] )
      { S7_Templates := "time_type := Time" } #statTonTime[190].TON(pt := #delayTime, et =>)
      Move(in := #STEP_IDLE, out1 => "Unit1.Em2.ControlNodes".jrOutPnPLeft.sequence.status.nextStep)
   END_RUNG
   // the same network as SCL:
   "Unit1.Em2.ControlNodes".jrOutPnPLeft."step".action1[190] := ("Unit1.Em2.ControlNodes".jrOutPnPLeft.sequence.status.currentStep = #JOB_1_STEP_90) AND "Unit1.Em2.ControlNodes".jrOutPnPLeft.sequence.status.seqActive;
   "Unit1.Em2.ControlNodes".jrOutPnPLeft."step".transition1[190] := ("Unit1.Em2.ControlNodes".jrOutPnPLeft.sequence.status.currentStep = #JOB_1_STEP_90) AND "Unit1.Em2.ControlNodes".jrOutPnPLeft.sequence.status.seqActive AND "Unit1.Em2.ControlNodes".cm.softcam.jrOutPnPLeftAxisX.pos00_wait.inPos AND "Unit1.Em2.ControlNodes".cm.softcam.jrOutPnPLeftAxisZ.pos00_wait.inPos AND ("Unit1.Em2.ControlNodes".cmJROutPnPLeftClampOpenClose.monitoring.inHomePos OR "Unit1.Em2.ControlNodes".cmJROutPnPLeftClampOpenClose.monitoring.inWorkPos);
   #statTonTime[190].TON(IN := ("Unit1.Em2.ControlNodes".jrOutPnPLeft.sequence.status.currentStep = #JOB_1_STEP_90) AND "Unit1.Em2.ControlNodes".jrOutPnPLeft.sequence.status.seqActive AND "Unit1.Em2.ControlNodes".jrOutPnPLeft."step".transition1[190],
                         PT := #delayTime);
   IF #statTonTime[190].Q THEN
       "Unit1.Em2.ControlNodes".jrOutPnPLeft.sequence.status.nextStep := #STEP_IDLE;
   END_IF;
END_REGION

REGION Network 13: *************** JOB[2] JR GET STACK-1=AUTO *************************
END_REGION

REGION Network 14: Step[201] : JOB[2] Condition
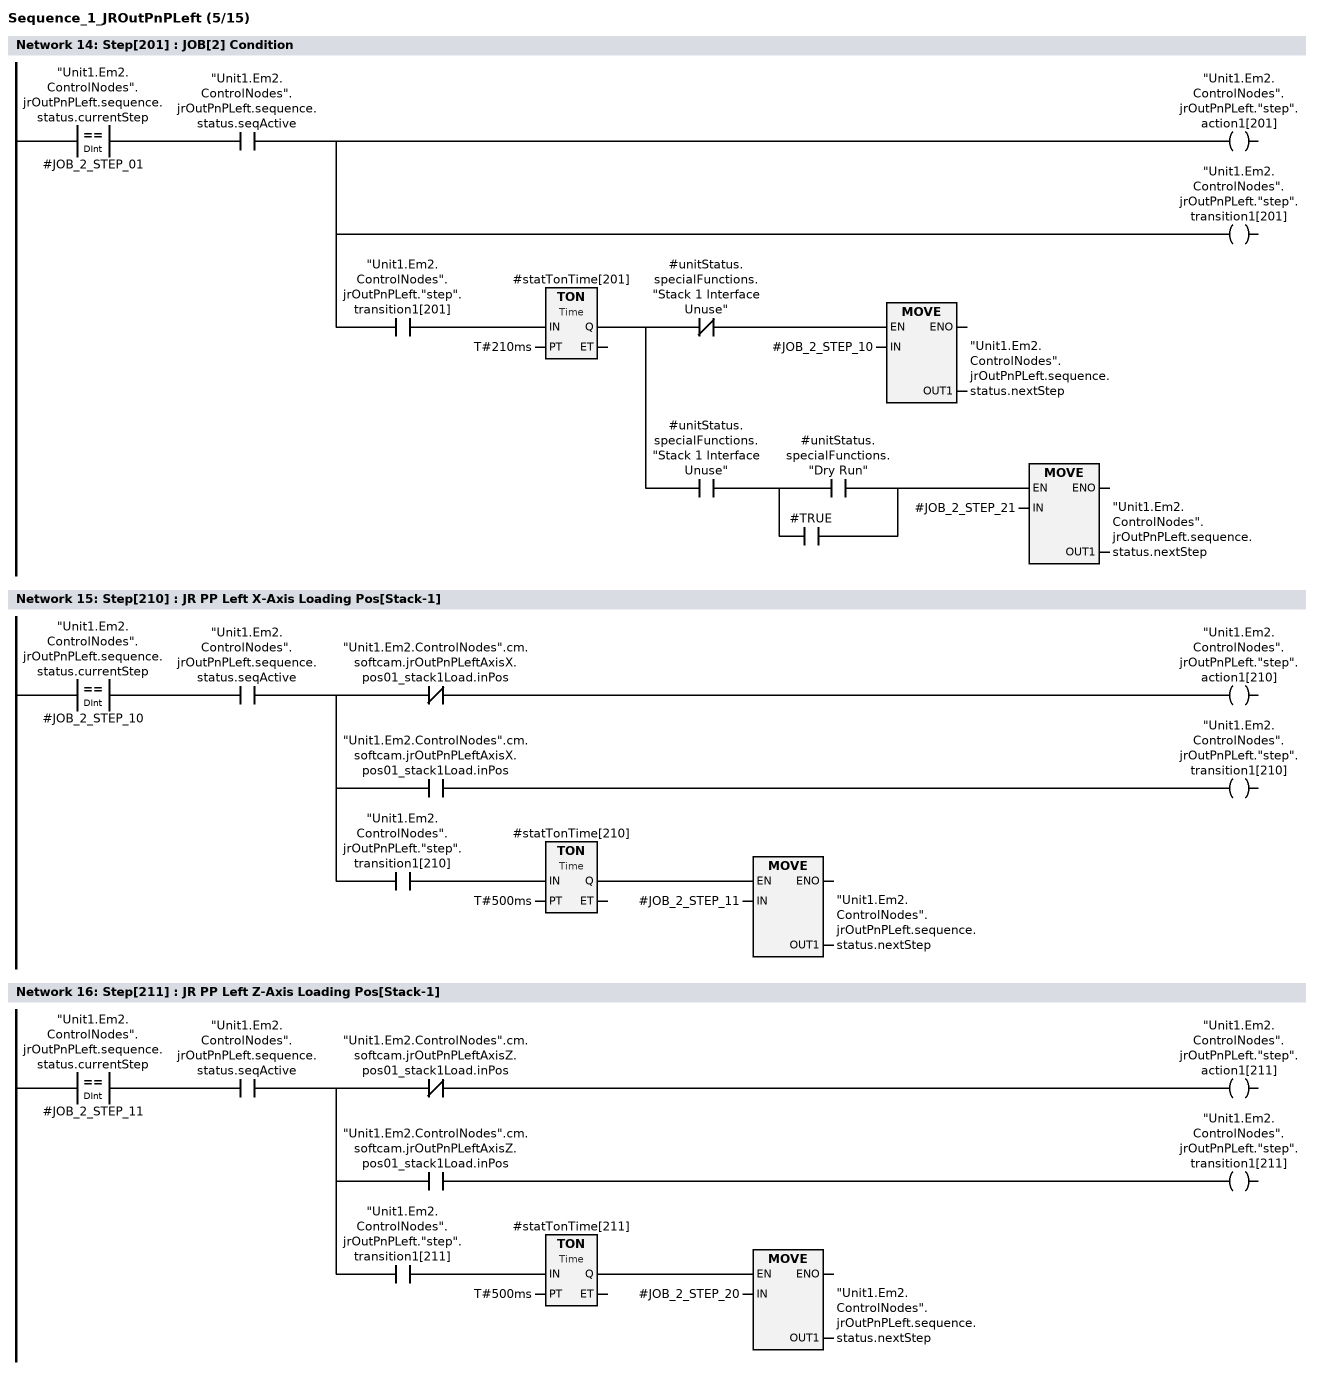
   RUNG wire#powerrail
      { S7_Templates := "SrcType := DInt" } EQ_Contact(in1 := "Unit1.Em2.ControlNodes".jrOutPnPLeft.sequence.status.currentStep, in2 := #JOB_2_STEP_01)
      Contact( "Unit1.Em2.ControlNodes".jrOutPnPLeft.sequence.status.seqActive )
      wire#w1
      Coil( "Unit1.Em2.ControlNodes".jrOutPnPLeft."step".action1[201] )
   END_RUNG
   RUNG wire#w1
      Coil( "Unit1.Em2.ControlNodes".jrOutPnPLeft."step".transition1[201] )
   END_RUNG
   RUNG wire#w1
      Contact( "Unit1.Em2.ControlNodes".jrOutPnPLeft."step".transition1[201] )
      { S7_Templates := "time_type := Time" } #statTonTime[201].TON(pt := T#210ms, et =>)
      wire#w2
      I_Contact( #unitStatus.specialFunctions."Stack 1 lnterface Unuse" )
      Move(in := #JOB_2_STEP_10, out1 => "Unit1.Em2.ControlNodes".jrOutPnPLeft.sequence.status.nextStep)
   END_RUNG
   RUNG wire#w2
      Contact( #unitStatus.specialFunctions."Stack 1 lnterface Unuse" )
      wire#w3
      Contact( #unitStatus.specialFunctions."Dry Run" )
      wire#w4
      Move(in := #JOB_2_STEP_21, out1 => "Unit1.Em2.ControlNodes".jrOutPnPLeft.sequence.status.nextStep)
   END_RUNG
   RUNG wire#w3
      Contact( #TRUE )
   END_RUNG wire#w4
   // the same network as SCL:
   "Unit1.Em2.ControlNodes".jrOutPnPLeft."step".action1[201] := ("Unit1.Em2.ControlNodes".jrOutPnPLeft.sequence.status.currentStep = #JOB_2_STEP_01) AND "Unit1.Em2.ControlNodes".jrOutPnPLeft.sequence.status.seqActive;
   "Unit1.Em2.ControlNodes".jrOutPnPLeft."step".transition1[201] := ("Unit1.Em2.ControlNodes".jrOutPnPLeft.sequence.status.currentStep = #JOB_2_STEP_01) AND "Unit1.Em2.ControlNodes".jrOutPnPLeft.sequence.status.seqActive;
   #statTonTime[201].TON(IN := ("Unit1.Em2.ControlNodes".jrOutPnPLeft.sequence.status.currentStep = #JOB_2_STEP_01) AND "Unit1.Em2.ControlNodes".jrOutPnPLeft.sequence.status.seqActive AND "Unit1.Em2.ControlNodes".jrOutPnPLeft."step".transition1[201],
                         PT := T#210ms);
   IF #statTonTime[201].Q AND NOT #unitStatus.specialFunctions."Stack 1 lnterface Unuse" THEN
       "Unit1.Em2.ControlNodes".jrOutPnPLeft.sequence.status.nextStep := #JOB_2_STEP_10;
   END_IF;
   IF #statTonTime[201].Q AND #unitStatus.specialFunctions."Stack 1 lnterface Unuse" AND (#unitStatus.specialFunctions."Dry Run" OR #TRUE) THEN
       "Unit1.Em2.ControlNodes".jrOutPnPLeft.sequence.status.nextStep := #JOB_2_STEP_21;
   END_IF;
END_REGION

REGION Network 15: Step[210] : JR PP Left X-Axis Loading Pos[Stack-1]
   RUNG wire#powerrail
      { S7_Templates := "SrcType := DInt" } EQ_Contact(in1 := "Unit1.Em2.ControlNodes".jrOutPnPLeft.sequence.status.currentStep, in2 := #JOB_2_STEP_10)
      Contact( "Unit1.Em2.ControlNodes".jrOutPnPLeft.sequence.status.seqActive )
      wire#w1
      I_Contact( "Unit1.Em2.ControlNodes".cm.softcam.jrOutPnPLeftAxisX.pos01_stack1Load.inPos )
      Coil( "Unit1.Em2.ControlNodes".jrOutPnPLeft."step".action1[210] )
   END_RUNG
   RUNG wire#w1
      Contact( "Unit1.Em2.ControlNodes".cm.softcam.jrOutPnPLeftAxisX.pos01_stack1Load.inPos )
      Coil( "Unit1.Em2.ControlNodes".jrOutPnPLeft."step".transition1[210] )
   END_RUNG
   RUNG wire#w1
      Contact( "Unit1.Em2.ControlNodes".jrOutPnPLeft."step".transition1[210] )
      { S7_Templates := "time_type := Time" } #statTonTime[210].TON(pt := T#500ms, et =>)
      Move(in := #JOB_2_STEP_11, out1 => "Unit1.Em2.ControlNodes".jrOutPnPLeft.sequence.status.nextStep)
   END_RUNG
   // the same network as SCL:
   #_w1 := ("Unit1.Em2.ControlNodes".jrOutPnPLeft.sequence.status.currentStep = #JOB_2_STEP_10) AND "Unit1.Em2.ControlNodes".jrOutPnPLeft.sequence.status.seqActive;
   "Unit1.Em2.ControlNodes".jrOutPnPLeft."step".action1[210] := #_w1 AND NOT "Unit1.Em2.ControlNodes".cm.softcam.jrOutPnPLeftAxisX.pos01_stack1Load.inPos;
   "Unit1.Em2.ControlNodes".jrOutPnPLeft."step".transition1[210] := #_w1 AND "Unit1.Em2.ControlNodes".cm.softcam.jrOutPnPLeftAxisX.pos01_stack1Load.inPos;
   #statTonTime[210].TON(IN := #_w1 AND "Unit1.Em2.ControlNodes".jrOutPnPLeft."step".transition1[210],
                         PT := T#500ms);
   IF #statTonTime[210].Q THEN
       "Unit1.Em2.ControlNodes".jrOutPnPLeft.sequence.status.nextStep := #JOB_2_STEP_11;
   END_IF;
END_REGION

REGION Network 16: Step[211] : JR PP Left Z-Axis Loading Pos[Stack-1]
   RUNG wire#powerrail
      { S7_Templates := "SrcType := DInt" } EQ_Contact(in1 := "Unit1.Em2.ControlNodes".jrOutPnPLeft.sequence.status.currentStep, in2 := #JOB_2_STEP_11)
      Contact( "Unit1.Em2.ControlNodes".jrOutPnPLeft.sequence.status.seqActive )
      wire#w1
      I_Contact( "Unit1.Em2.ControlNodes".cm.softcam.jrOutPnPLeftAxisZ.pos01_stack1Load.inPos )
      Coil( "Unit1.Em2.ControlNodes".jrOutPnPLeft."step".action1[211] )
   END_RUNG
   RUNG wire#w1
      Contact( "Unit1.Em2.ControlNodes".cm.softcam.jrOutPnPLeftAxisZ.pos01_stack1Load.inPos )
      Coil( "Unit1.Em2.ControlNodes".jrOutPnPLeft."step".transition1[211] )
   END_RUNG
   RUNG wire#w1
      Contact( "Unit1.Em2.ControlNodes".jrOutPnPLeft."step".transition1[211] )
      { S7_Templates := "time_type := Time" } #statTonTime[211].TON(pt := T#500ms, et =>)
      Move(in := #JOB_2_STEP_20, out1 => "Unit1.Em2.ControlNodes".jrOutPnPLeft.sequence.status.nextStep)
   END_RUNG
   // the same network as SCL:
   #_w1 := ("Unit1.Em2.ControlNodes".jrOutPnPLeft.sequence.status.currentStep = #JOB_2_STEP_11) AND "Unit1.Em2.ControlNodes".jrOutPnPLeft.sequence.status.seqActive;
   "Unit1.Em2.ControlNodes".jrOutPnPLeft."step".action1[211] := #_w1 AND NOT "Unit1.Em2.ControlNodes".cm.softcam.jrOutPnPLeftAxisZ.pos01_stack1Load.inPos;
   "Unit1.Em2.ControlNodes".jrOutPnPLeft."step".transition1[211] := #_w1 AND "Unit1.Em2.ControlNodes".cm.softcam.jrOutPnPLeftAxisZ.pos01_stack1Load.inPos;
   #statTonTime[211].TON(IN := #_w1 AND "Unit1.Em2.ControlNodes".jrOutPnPLeft."step".transition1[211],
                         PT := T#500ms);
   IF #statTonTime[211].Q THEN
       "Unit1.Em2.ControlNodes".jrOutPnPLeft.sequence.status.nextStep := #JOB_2_STEP_20;
   END_IF;
END_REGION

REGION Network 17: Step[220] : JR PP Left [OnPosition Unloading] => Stack #1
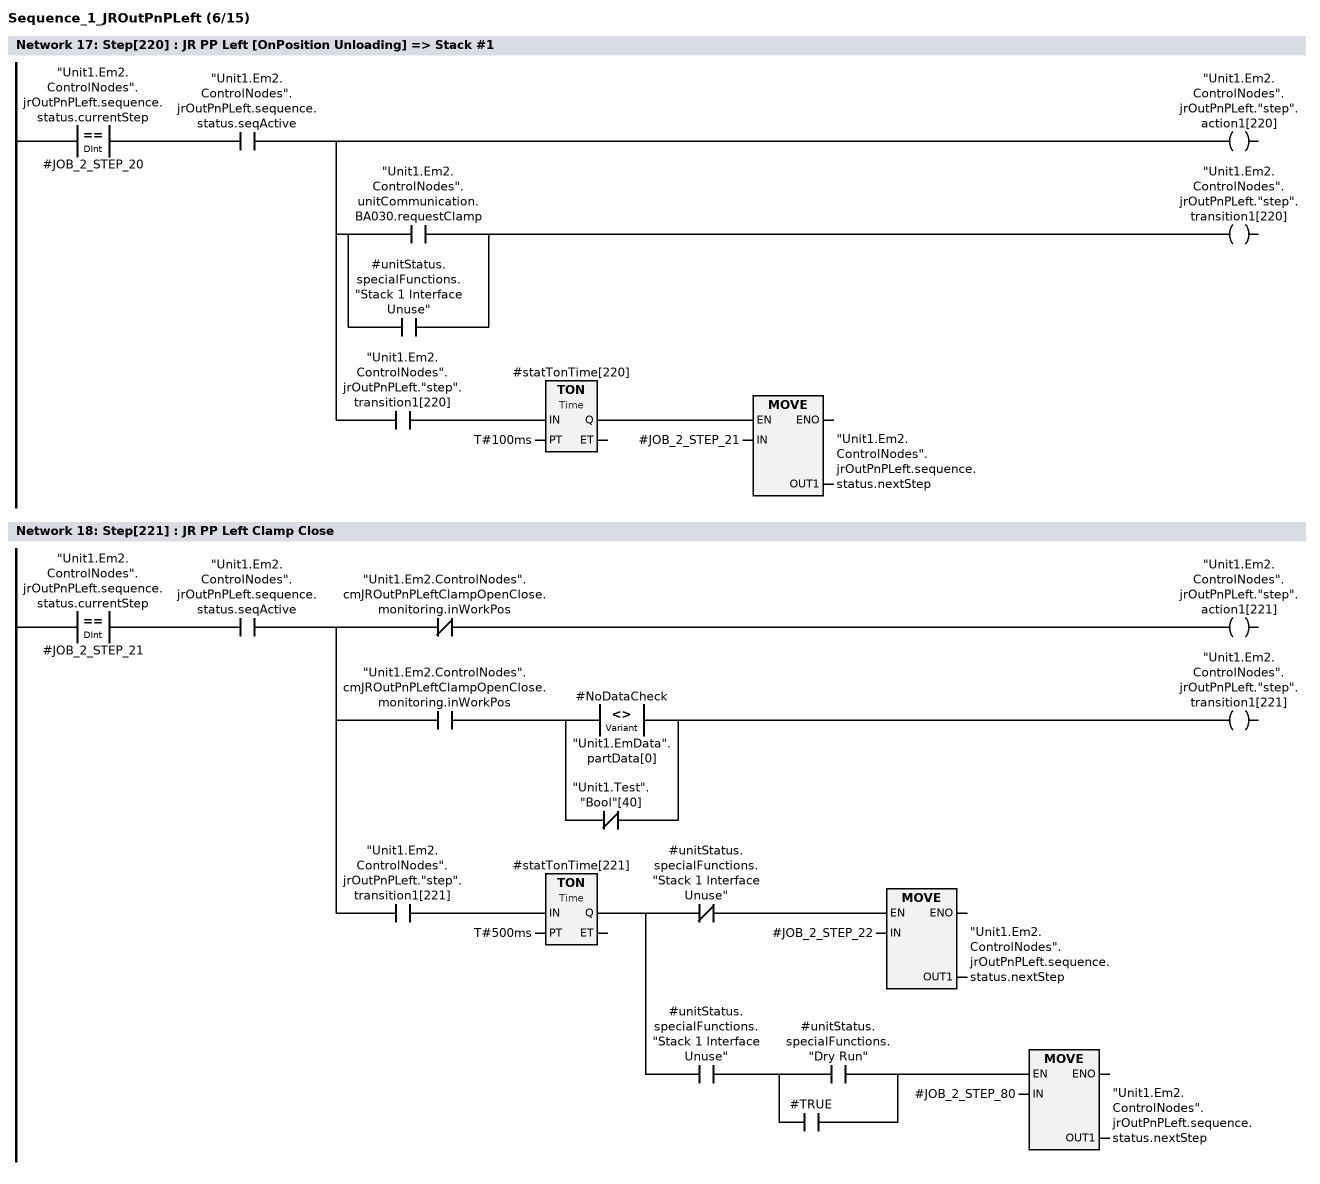
   RUNG wire#powerrail
      { S7_Templates := "SrcType := DInt" } EQ_Contact(in1 := "Unit1.Em2.ControlNodes".jrOutPnPLeft.sequence.status.currentStep, in2 := #JOB_2_STEP_20)
      Contact( "Unit1.Em2.ControlNodes".jrOutPnPLeft.sequence.status.seqActive )
      wire#w1
      Coil( "Unit1.Em2.ControlNodes".jrOutPnPLeft."step".action1[220] )
   END_RUNG
   RUNG wire#w1
      Contact( "Unit1.Em2.ControlNodes".unitCommunication.BA030.requestClamp )
      wire#w2
      Coil( "Unit1.Em2.ControlNodes".jrOutPnPLeft."step".transition1[220] )
   END_RUNG
   RUNG wire#w1
      Contact( #unitStatus.specialFunctions."Stack 1 lnterface Unuse" )
   END_RUNG wire#w2
   RUNG wire#w1
      Contact( "Unit1.Em2.ControlNodes".jrOutPnPLeft."step".transition1[220] )
      { S7_Templates := "time_type := Time" } #statTonTime[220].TON(pt := T#100ms, et =>)
      Move(in := #JOB_2_STEP_21, out1 => "Unit1.Em2.ControlNodes".jrOutPnPLeft.sequence.status.nextStep)
   END_RUNG
   // the same network as SCL:
   "Unit1.Em2.ControlNodes".jrOutPnPLeft."step".action1[220] := ("Unit1.Em2.ControlNodes".jrOutPnPLeft.sequence.status.currentStep = #JOB_2_STEP_20) AND "Unit1.Em2.ControlNodes".jrOutPnPLeft.sequence.status.seqActive;
   "Unit1.Em2.ControlNodes".jrOutPnPLeft."step".transition1[220] := ("Unit1.Em2.ControlNodes".jrOutPnPLeft.sequence.status.currentStep = #JOB_2_STEP_20) AND "Unit1.Em2.ControlNodes".jrOutPnPLeft.sequence.status.seqActive AND ("Unit1.Em2.ControlNodes".unitCommunication.BA030.requestClamp OR #unitStatus.specialFunctions."Stack 1 lnterface Unuse");
   #statTonTime[220].TON(IN := ("Unit1.Em2.ControlNodes".jrOutPnPLeft.sequence.status.currentStep = #JOB_2_STEP_20) AND "Unit1.Em2.ControlNodes".jrOutPnPLeft.sequence.status.seqActive AND "Unit1.Em2.ControlNodes".jrOutPnPLeft."step".transition1[220],
                         PT := T#100ms);
   IF #statTonTime[220].Q THEN
       "Unit1.Em2.ControlNodes".jrOutPnPLeft.sequence.status.nextStep := #JOB_2_STEP_21;
   END_IF;
END_REGION

REGION Network 18: Step[221] : JR PP Left Clamp Close
   RUNG wire#powerrail
      { S7_Templates := "SrcType := DInt" } EQ_Contact(in1 := "Unit1.Em2.ControlNodes".jrOutPnPLeft.sequence.status.currentStep, in2 := #JOB_2_STEP_21)
      Contact( "Unit1.Em2.ControlNodes".jrOutPnPLeft.sequence.status.seqActive )
      wire#w1
      I_Contact( "Unit1.Em2.ControlNodes".cmJROutPnPLeftClampOpenClose.monitoring.inWorkPos )
      Coil( "Unit1.Em2.ControlNodes".jrOutPnPLeft."step".action1[221] )
   END_RUNG
   RUNG wire#w1
      Contact( "Unit1.Em2.ControlNodes".cmJROutPnPLeftClampOpenClose.monitoring.inWorkPos )
      wire#w2
      { S7_Templates := "SrcType := Variant" } NE_Contact(in1 := #NoDataCheck, in2 := "Unit1.EmData".partData[0])
      wire#w3
      Coil( "Unit1.Em2.ControlNodes".jrOutPnPLeft."step".transition1[221] )
   END_RUNG
   RUNG wire#w2
      I_Contact( "Unit1.Test"."Bool"[40] )
   END_RUNG wire#w3
   RUNG wire#w1
      Contact( "Unit1.Em2.ControlNodes".jrOutPnPLeft."step".transition1[221] )
      { S7_Templates := "time_type := Time" } #statTonTime[221].TON(pt := T#500ms, et =>)
      wire#w4
      I_Contact( #unitStatus.specialFunctions."Stack 1 lnterface Unuse" )
      Move(in := #JOB_2_STEP_22, out1 => "Unit1.Em2.ControlNodes".jrOutPnPLeft.sequence.status.nextStep)
   END_RUNG
   RUNG wire#w4
      Contact( #unitStatus.specialFunctions."Stack 1 lnterface Unuse" )
      wire#w5
      Contact( #unitStatus.specialFunctions."Dry Run" )
      wire#w6
      Move(in := #JOB_2_STEP_80, out1 => "Unit1.Em2.ControlNodes".jrOutPnPLeft.sequence.status.nextStep)
   END_RUNG
   RUNG wire#w5
      Contact( #TRUE )
   END_RUNG wire#w6
   // the same network as SCL:
   #_w1 := ("Unit1.Em2.ControlNodes".jrOutPnPLeft.sequence.status.currentStep = #JOB_2_STEP_21) AND "Unit1.Em2.ControlNodes".jrOutPnPLeft.sequence.status.seqActive;
   "Unit1.Em2.ControlNodes".jrOutPnPLeft."step".action1[221] := #_w1 AND NOT "Unit1.Em2.ControlNodes".cmJROutPnPLeftClampOpenClose.monitoring.inWorkPos;
   "Unit1.Em2.ControlNodes".jrOutPnPLeft."step".transition1[221] := #_w1 AND "Unit1.Em2.ControlNodes".cmJROutPnPLeftClampOpenClose.monitoring.inWorkPos AND ((#NoDataCheck <> "Unit1.EmData".partData[0]) OR NOT "Unit1.Test"."Bool"[40]);
   #statTonTime[221].TON(IN := #_w1 AND "Unit1.Em2.ControlNodes".jrOutPnPLeft."step".transition1[221],
                         PT := T#500ms);
   IF #statTonTime[221].Q AND NOT #unitStatus.specialFunctions."Stack 1 lnterface Unuse" THEN
       "Unit1.Em2.ControlNodes".jrOutPnPLeft.sequence.status.nextStep := #JOB_2_STEP_22;
   END_IF;
   IF #statTonTime[221].Q AND #unitStatus.specialFunctions."Stack 1 lnterface Unuse" AND (#unitStatus.specialFunctions."Dry Run" OR #TRUE) THEN
       "Unit1.Em2.ControlNodes".jrOutPnPLeft.sequence.status.nextStep := #JOB_2_STEP_80;
   END_IF;
END_REGION

REGION Network 19: Step[222] : JR PP Left [Request Unclamp] => Stack #1
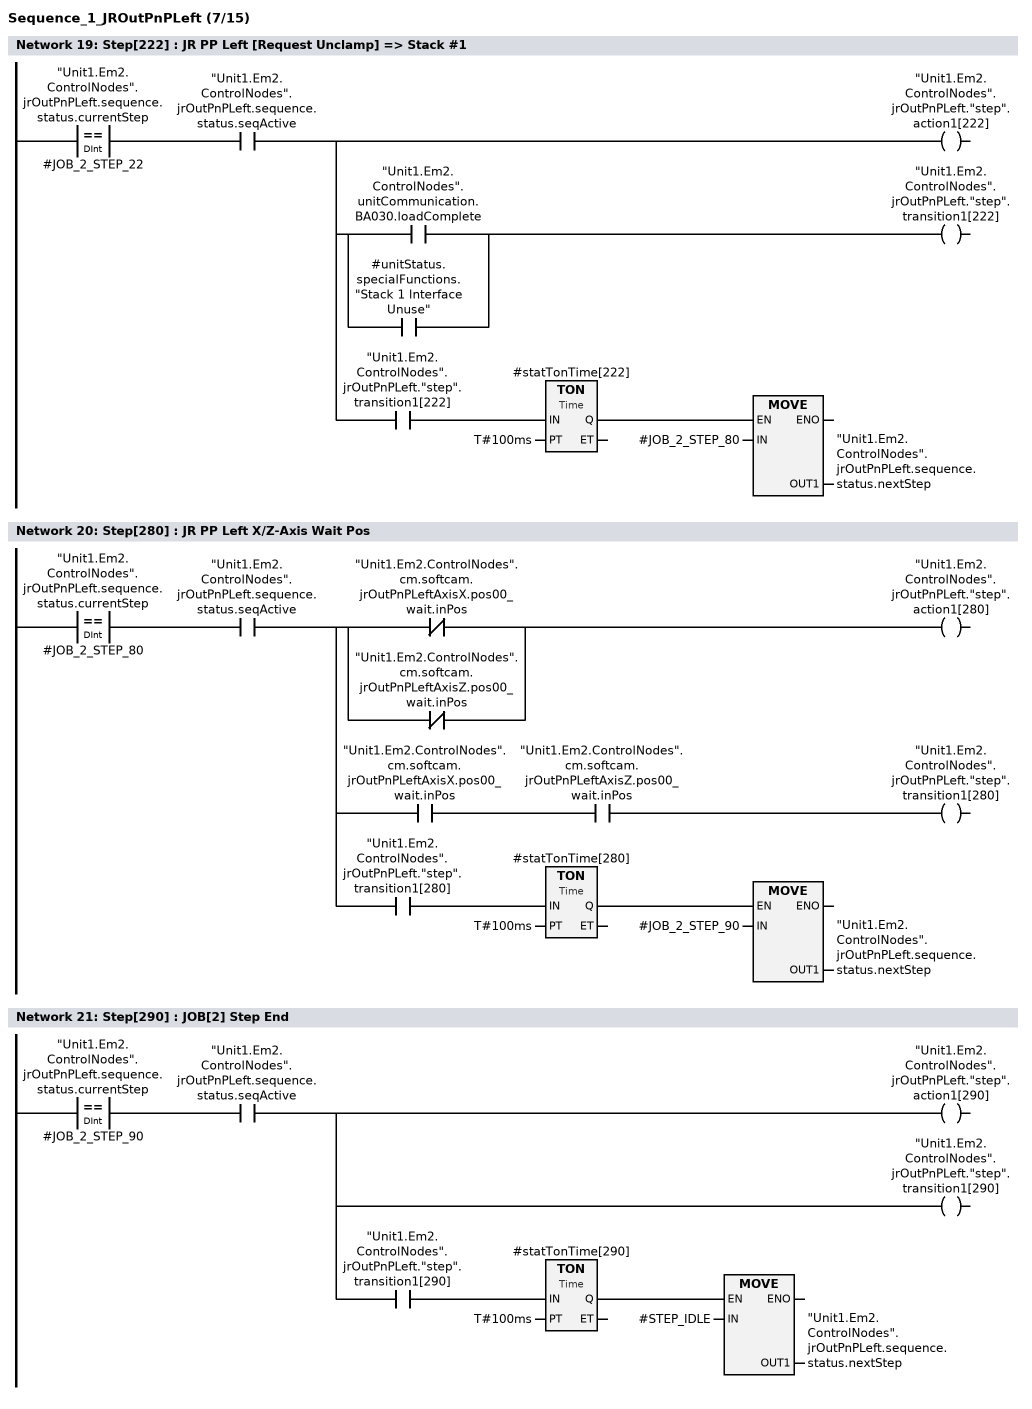
   RUNG wire#powerrail
      { S7_Templates := "SrcType := DInt" } EQ_Contact(in1 := "Unit1.Em2.ControlNodes".jrOutPnPLeft.sequence.status.currentStep, in2 := #JOB_2_STEP_22)
      Contact( "Unit1.Em2.ControlNodes".jrOutPnPLeft.sequence.status.seqActive )
      wire#w1
      Coil( "Unit1.Em2.ControlNodes".jrOutPnPLeft."step".action1[222] )
   END_RUNG
   RUNG wire#w1
      Contact( "Unit1.Em2.ControlNodes".unitCommunication.BA030.loadComplete )
      wire#w2
      Coil( "Unit1.Em2.ControlNodes".jrOutPnPLeft."step".transition1[222] )
   END_RUNG
   RUNG wire#w1
      Contact( #unitStatus.specialFunctions."Stack 1 lnterface Unuse" )
   END_RUNG wire#w2
   RUNG wire#w1
      Contact( "Unit1.Em2.ControlNodes".jrOutPnPLeft."step".transition1[222] )
      { S7_Templates := "time_type := Time" } #statTonTime[222].TON(pt := T#100ms, et =>)
      Move(in := #JOB_2_STEP_80, out1 => "Unit1.Em2.ControlNodes".jrOutPnPLeft.sequence.status.nextStep)
   END_RUNG
   // the same network as SCL:
   "Unit1.Em2.ControlNodes".jrOutPnPLeft."step".action1[222] := ("Unit1.Em2.ControlNodes".jrOutPnPLeft.sequence.status.currentStep = #JOB_2_STEP_22) AND "Unit1.Em2.ControlNodes".jrOutPnPLeft.sequence.status.seqActive;
   "Unit1.Em2.ControlNodes".jrOutPnPLeft."step".transition1[222] := ("Unit1.Em2.ControlNodes".jrOutPnPLeft.sequence.status.currentStep = #JOB_2_STEP_22) AND "Unit1.Em2.ControlNodes".jrOutPnPLeft.sequence.status.seqActive AND ("Unit1.Em2.ControlNodes".unitCommunication.BA030.loadComplete OR #unitStatus.specialFunctions."Stack 1 lnterface Unuse");
   #statTonTime[222].TON(IN := ("Unit1.Em2.ControlNodes".jrOutPnPLeft.sequence.status.currentStep = #JOB_2_STEP_22) AND "Unit1.Em2.ControlNodes".jrOutPnPLeft.sequence.status.seqActive AND "Unit1.Em2.ControlNodes".jrOutPnPLeft."step".transition1[222],
                         PT := T#100ms);
   IF #statTonTime[222].Q THEN
       "Unit1.Em2.ControlNodes".jrOutPnPLeft.sequence.status.nextStep := #JOB_2_STEP_80;
   END_IF;
END_REGION

REGION Network 20: Step[280] : JR PP Left X/Z-Axis Wait Pos
   RUNG wire#powerrail
      { S7_Templates := "SrcType := DInt" } EQ_Contact(in1 := "Unit1.Em2.ControlNodes".jrOutPnPLeft.sequence.status.currentStep, in2 := #JOB_2_STEP_80)
      Contact( "Unit1.Em2.ControlNodes".jrOutPnPLeft.sequence.status.seqActive )
      wire#w1
      I_Contact( "Unit1.Em2.ControlNodes".cm.softcam.jrOutPnPLeftAxisX.pos00_wait.inPos )
      wire#w2
      Coil( "Unit1.Em2.ControlNodes".jrOutPnPLeft."step".action1[280] )
   END_RUNG
   RUNG wire#w1
      I_Contact( "Unit1.Em2.ControlNodes".cm.softcam.jrOutPnPLeftAxisZ.pos00_wait.inPos )
   END_RUNG wire#w2
   RUNG wire#w1
      Contact( "Unit1.Em2.ControlNodes".cm.softcam.jrOutPnPLeftAxisX.pos00_wait.inPos )
      Contact( "Unit1.Em2.ControlNodes".cm.softcam.jrOutPnPLeftAxisZ.pos00_wait.inPos )
      Coil( "Unit1.Em2.ControlNodes".jrOutPnPLeft."step".transition1[280] )
   END_RUNG
   RUNG wire#w1
      Contact( "Unit1.Em2.ControlNodes".jrOutPnPLeft."step".transition1[280] )
      { S7_Templates := "time_type := Time" } #statTonTime[280].TON(pt := T#100ms, et =>)
      Move(in := #JOB_2_STEP_90, out1 => "Unit1.Em2.ControlNodes".jrOutPnPLeft.sequence.status.nextStep)
   END_RUNG
   // the same network as SCL:
   #_w1 := ("Unit1.Em2.ControlNodes".jrOutPnPLeft.sequence.status.currentStep = #JOB_2_STEP_80) AND "Unit1.Em2.ControlNodes".jrOutPnPLeft.sequence.status.seqActive;
   "Unit1.Em2.ControlNodes".jrOutPnPLeft."step".action1[280] := #_w1 AND (NOT "Unit1.Em2.ControlNodes".cm.softcam.jrOutPnPLeftAxisX.pos00_wait.inPos OR NOT "Unit1.Em2.ControlNodes".cm.softcam.jrOutPnPLeftAxisZ.pos00_wait.inPos);
   "Unit1.Em2.ControlNodes".jrOutPnPLeft."step".transition1[280] := #_w1 AND "Unit1.Em2.ControlNodes".cm.softcam.jrOutPnPLeftAxisX.pos00_wait.inPos AND "Unit1.Em2.ControlNodes".cm.softcam.jrOutPnPLeftAxisZ.pos00_wait.inPos;
   #statTonTime[280].TON(IN := #_w1 AND "Unit1.Em2.ControlNodes".jrOutPnPLeft."step".transition1[280],
                         PT := T#100ms);
   IF #statTonTime[280].Q THEN
       "Unit1.Em2.ControlNodes".jrOutPnPLeft.sequence.status.nextStep := #JOB_2_STEP_90;
   END_IF;
END_REGION

REGION Network 21: Step[290] : JOB[2] Step End
   RUNG wire#powerrail
      { S7_Templates := "SrcType := DInt" } EQ_Contact(in1 := "Unit1.Em2.ControlNodes".jrOutPnPLeft.sequence.status.currentStep, in2 := #JOB_2_STEP_90)
      Contact( "Unit1.Em2.ControlNodes".jrOutPnPLeft.sequence.status.seqActive )
      wire#w1
      Coil( "Unit1.Em2.ControlNodes".jrOutPnPLeft."step".action1[290] )
   END_RUNG
   RUNG wire#w1
      Coil( "Unit1.Em2.ControlNodes".jrOutPnPLeft."step".transition1[290] )
   END_RUNG
   RUNG wire#w1
      Contact( "Unit1.Em2.ControlNodes".jrOutPnPLeft."step".transition1[290] )
      { S7_Templates := "time_type := Time" } #statTonTime[290].TON(pt := T#100ms, et =>)
      Move(in := #STEP_IDLE, out1 => "Unit1.Em2.ControlNodes".jrOutPnPLeft.sequence.status.nextStep)
   END_RUNG
   // the same network as SCL:
   "Unit1.Em2.ControlNodes".jrOutPnPLeft."step".action1[290] := ("Unit1.Em2.ControlNodes".jrOutPnPLeft.sequence.status.currentStep = #JOB_2_STEP_90) AND "Unit1.Em2.ControlNodes".jrOutPnPLeft.sequence.status.seqActive;
   "Unit1.Em2.ControlNodes".jrOutPnPLeft."step".transition1[290] := ("Unit1.Em2.ControlNodes".jrOutPnPLeft.sequence.status.currentStep = #JOB_2_STEP_90) AND "Unit1.Em2.ControlNodes".jrOutPnPLeft.sequence.status.seqActive;
   #statTonTime[290].TON(IN := ("Unit1.Em2.ControlNodes".jrOutPnPLeft.sequence.status.currentStep = #JOB_2_STEP_90) AND "Unit1.Em2.ControlNodes".jrOutPnPLeft.sequence.status.seqActive AND "Unit1.Em2.ControlNodes".jrOutPnPLeft."step".transition1[290],
                         PT := T#100ms);
   IF #statTonTime[290].Q THEN
       "Unit1.Em2.ControlNodes".jrOutPnPLeft.sequence.status.nextStep := #STEP_IDLE;
   END_IF;
END_REGION

REGION Network 22: *************** JOB[3] JR GET STACK-2=AUTO *************************
END_REGION

REGION Network 23: Step[301] : JOB[3] Condition
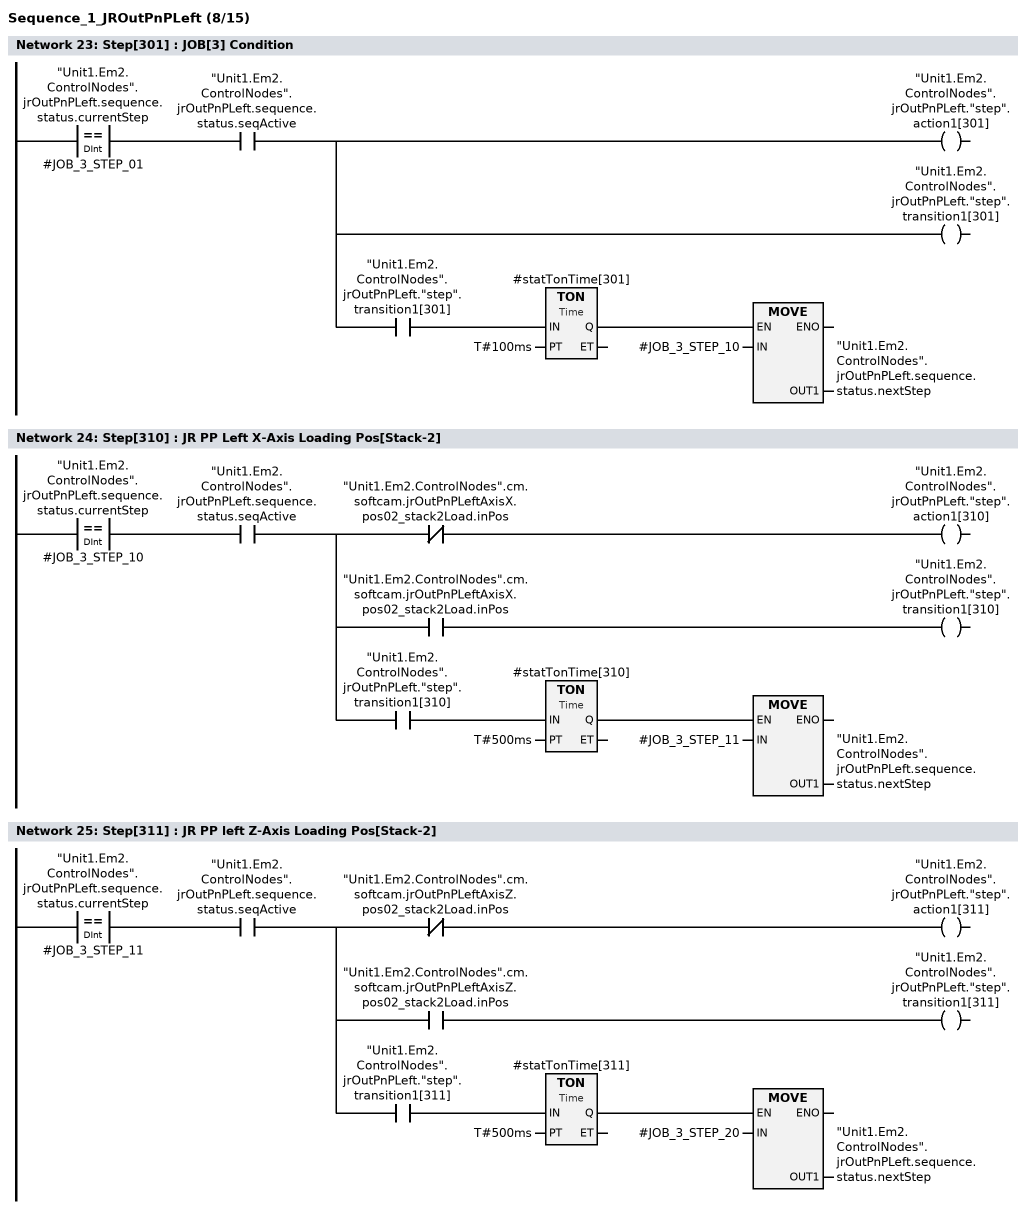
   RUNG wire#powerrail
      { S7_Templates := "SrcType := DInt" } EQ_Contact(in1 := "Unit1.Em2.ControlNodes".jrOutPnPLeft.sequence.status.currentStep, in2 := #JOB_3_STEP_01)
      Contact( "Unit1.Em2.ControlNodes".jrOutPnPLeft.sequence.status.seqActive )
      wire#w1
      Coil( "Unit1.Em2.ControlNodes".jrOutPnPLeft."step".action1[301] )
   END_RUNG
   RUNG wire#w1
      Coil( "Unit1.Em2.ControlNodes".jrOutPnPLeft."step".transition1[301] )
   END_RUNG
   RUNG wire#w1
      Contact( "Unit1.Em2.ControlNodes".jrOutPnPLeft."step".transition1[301] )
      { S7_Templates := "time_type := Time" } #statTonTime[301].TON(pt := T#100ms, et =>)
      Move(in := #JOB_3_STEP_10, out1 => "Unit1.Em2.ControlNodes".jrOutPnPLeft.sequence.status.nextStep)
   END_RUNG
   // the same network as SCL:
   "Unit1.Em2.ControlNodes".jrOutPnPLeft."step".action1[301] := ("Unit1.Em2.ControlNodes".jrOutPnPLeft.sequence.status.currentStep = #JOB_3_STEP_01) AND "Unit1.Em2.ControlNodes".jrOutPnPLeft.sequence.status.seqActive;
   "Unit1.Em2.ControlNodes".jrOutPnPLeft."step".transition1[301] := ("Unit1.Em2.ControlNodes".jrOutPnPLeft.sequence.status.currentStep = #JOB_3_STEP_01) AND "Unit1.Em2.ControlNodes".jrOutPnPLeft.sequence.status.seqActive;
   #statTonTime[301].TON(IN := ("Unit1.Em2.ControlNodes".jrOutPnPLeft.sequence.status.currentStep = #JOB_3_STEP_01) AND "Unit1.Em2.ControlNodes".jrOutPnPLeft.sequence.status.seqActive AND "Unit1.Em2.ControlNodes".jrOutPnPLeft."step".transition1[301],
                         PT := T#100ms);
   IF #statTonTime[301].Q THEN
       "Unit1.Em2.ControlNodes".jrOutPnPLeft.sequence.status.nextStep := #JOB_3_STEP_10;
   END_IF;
END_REGION

REGION Network 24: Step[310] : JR PP Left X-Axis Loading Pos[Stack-2]
   RUNG wire#powerrail
      { S7_Templates := "SrcType := DInt" } EQ_Contact(in1 := "Unit1.Em2.ControlNodes".jrOutPnPLeft.sequence.status.currentStep, in2 := #JOB_3_STEP_10)
      Contact( "Unit1.Em2.ControlNodes".jrOutPnPLeft.sequence.status.seqActive )
      wire#w1
      I_Contact( "Unit1.Em2.ControlNodes".cm.softcam.jrOutPnPLeftAxisX.pos02_stack2Load.inPos )
      Coil( "Unit1.Em2.ControlNodes".jrOutPnPLeft."step".action1[310] )
   END_RUNG
   RUNG wire#w1
      Contact( "Unit1.Em2.ControlNodes".cm.softcam.jrOutPnPLeftAxisX.pos02_stack2Load.inPos )
      Coil( "Unit1.Em2.ControlNodes".jrOutPnPLeft."step".transition1[310] )
   END_RUNG
   RUNG wire#w1
      Contact( "Unit1.Em2.ControlNodes".jrOutPnPLeft."step".transition1[310] )
      { S7_Templates := "time_type := Time" } #statTonTime[310].TON(pt := T#500ms, et =>)
      Move(in := #JOB_3_STEP_11, out1 => "Unit1.Em2.ControlNodes".jrOutPnPLeft.sequence.status.nextStep)
   END_RUNG
   // the same network as SCL:
   #_w1 := ("Unit1.Em2.ControlNodes".jrOutPnPLeft.sequence.status.currentStep = #JOB_3_STEP_10) AND "Unit1.Em2.ControlNodes".jrOutPnPLeft.sequence.status.seqActive;
   "Unit1.Em2.ControlNodes".jrOutPnPLeft."step".action1[310] := #_w1 AND NOT "Unit1.Em2.ControlNodes".cm.softcam.jrOutPnPLeftAxisX.pos02_stack2Load.inPos;
   "Unit1.Em2.ControlNodes".jrOutPnPLeft."step".transition1[310] := #_w1 AND "Unit1.Em2.ControlNodes".cm.softcam.jrOutPnPLeftAxisX.pos02_stack2Load.inPos;
   #statTonTime[310].TON(IN := #_w1 AND "Unit1.Em2.ControlNodes".jrOutPnPLeft."step".transition1[310],
                         PT := T#500ms);
   IF #statTonTime[310].Q THEN
       "Unit1.Em2.ControlNodes".jrOutPnPLeft.sequence.status.nextStep := #JOB_3_STEP_11;
   END_IF;
END_REGION

REGION Network 25: Step[311] : JR PP left Z-Axis Loading Pos[Stack-2]
   RUNG wire#powerrail
      { S7_Templates := "SrcType := DInt" } EQ_Contact(in1 := "Unit1.Em2.ControlNodes".jrOutPnPLeft.sequence.status.currentStep, in2 := #JOB_3_STEP_11)
      Contact( "Unit1.Em2.ControlNodes".jrOutPnPLeft.sequence.status.seqActive )
      wire#w1
      I_Contact( "Unit1.Em2.ControlNodes".cm.softcam.jrOutPnPLeftAxisZ.pos02_stack2Load.inPos )
      Coil( "Unit1.Em2.ControlNodes".jrOutPnPLeft."step".action1[311] )
   END_RUNG
   RUNG wire#w1
      Contact( "Unit1.Em2.ControlNodes".cm.softcam.jrOutPnPLeftAxisZ.pos02_stack2Load.inPos )
      Coil( "Unit1.Em2.ControlNodes".jrOutPnPLeft."step".transition1[311] )
   END_RUNG
   RUNG wire#w1
      Contact( "Unit1.Em2.ControlNodes".jrOutPnPLeft."step".transition1[311] )
      { S7_Templates := "time_type := Time" } #statTonTime[311].TON(pt := T#500ms, et =>)
      Move(in := #JOB_3_STEP_20, out1 => "Unit1.Em2.ControlNodes".jrOutPnPLeft.sequence.status.nextStep)
   END_RUNG
   // the same network as SCL:
   #_w1 := ("Unit1.Em2.ControlNodes".jrOutPnPLeft.sequence.status.currentStep = #JOB_3_STEP_11) AND "Unit1.Em2.ControlNodes".jrOutPnPLeft.sequence.status.seqActive;
   "Unit1.Em2.ControlNodes".jrOutPnPLeft."step".action1[311] := #_w1 AND NOT "Unit1.Em2.ControlNodes".cm.softcam.jrOutPnPLeftAxisZ.pos02_stack2Load.inPos;
   "Unit1.Em2.ControlNodes".jrOutPnPLeft."step".transition1[311] := #_w1 AND "Unit1.Em2.ControlNodes".cm.softcam.jrOutPnPLeftAxisZ.pos02_stack2Load.inPos;
   #statTonTime[311].TON(IN := #_w1 AND "Unit1.Em2.ControlNodes".jrOutPnPLeft."step".transition1[311],
                         PT := T#500ms);
   IF #statTonTime[311].Q THEN
       "Unit1.Em2.ControlNodes".jrOutPnPLeft.sequence.status.nextStep := #JOB_3_STEP_20;
   END_IF;
END_REGION

REGION Network 26: Step[320] : JR PP Left [OnPosition Unloading] <= Stack #2
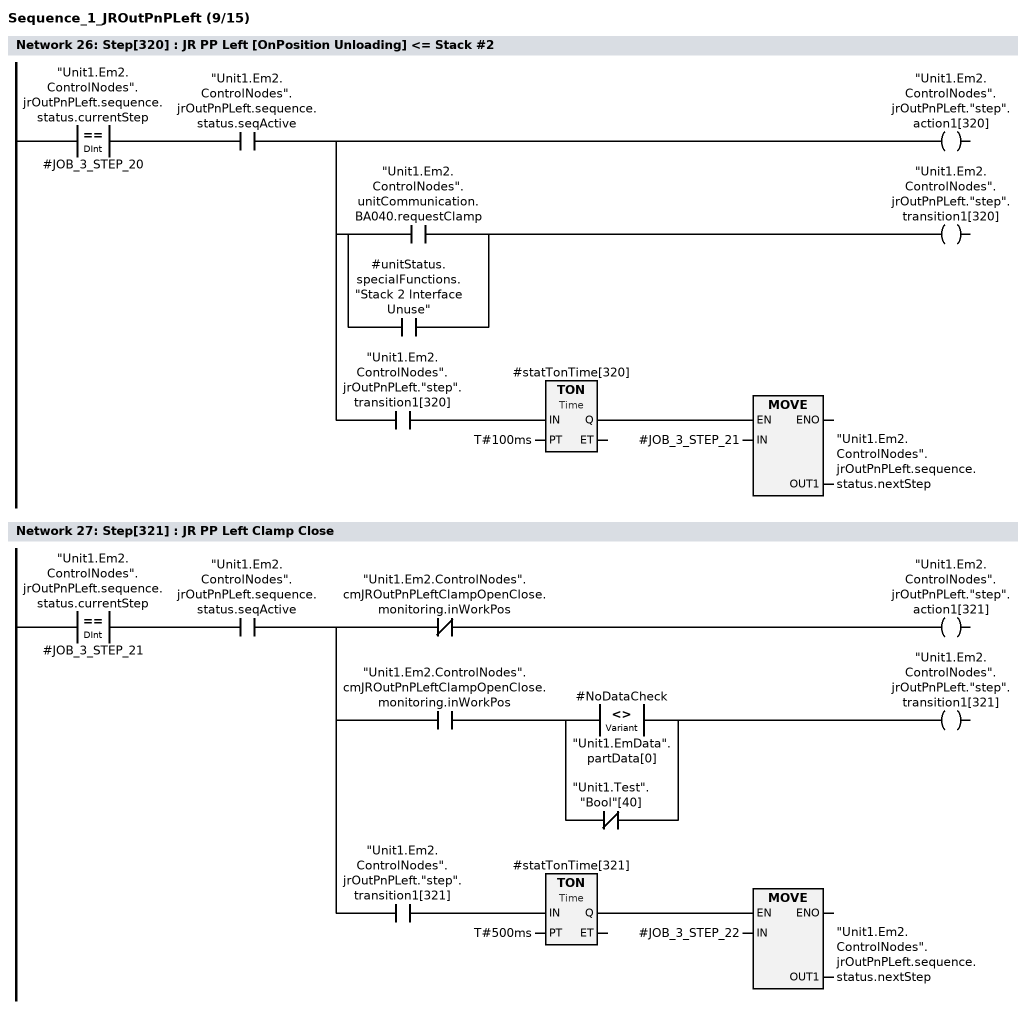
   RUNG wire#powerrail
      { S7_Templates := "SrcType := DInt" } EQ_Contact(in1 := "Unit1.Em2.ControlNodes".jrOutPnPLeft.sequence.status.currentStep, in2 := #JOB_3_STEP_20)
      Contact( "Unit1.Em2.ControlNodes".jrOutPnPLeft.sequence.status.seqActive )
      wire#w1
      Coil( "Unit1.Em2.ControlNodes".jrOutPnPLeft."step".action1[320] )
   END_RUNG
   RUNG wire#w1
      Contact( "Unit1.Em2.ControlNodes".unitCommunication.BA040.requestClamp )
      wire#w2
      Coil( "Unit1.Em2.ControlNodes".jrOutPnPLeft."step".transition1[320] )
   END_RUNG
   RUNG wire#w1
      Contact( #unitStatus.specialFunctions."Stack 2 lnterface Unuse" )
   END_RUNG wire#w2
   RUNG wire#w1
      Contact( "Unit1.Em2.ControlNodes".jrOutPnPLeft."step".transition1[320] )
      { S7_Templates := "time_type := Time" } #statTonTime[320].TON(pt := T#100ms, et =>)
      Move(in := #JOB_3_STEP_21, out1 => "Unit1.Em2.ControlNodes".jrOutPnPLeft.sequence.status.nextStep)
   END_RUNG
   // the same network as SCL:
   "Unit1.Em2.ControlNodes".jrOutPnPLeft."step".action1[320] := ("Unit1.Em2.ControlNodes".jrOutPnPLeft.sequence.status.currentStep = #JOB_3_STEP_20) AND "Unit1.Em2.ControlNodes".jrOutPnPLeft.sequence.status.seqActive;
   "Unit1.Em2.ControlNodes".jrOutPnPLeft."step".transition1[320] := ("Unit1.Em2.ControlNodes".jrOutPnPLeft.sequence.status.currentStep = #JOB_3_STEP_20) AND "Unit1.Em2.ControlNodes".jrOutPnPLeft.sequence.status.seqActive AND ("Unit1.Em2.ControlNodes".unitCommunication.BA040.requestClamp OR #unitStatus.specialFunctions."Stack 2 lnterface Unuse");
   #statTonTime[320].TON(IN := ("Unit1.Em2.ControlNodes".jrOutPnPLeft.sequence.status.currentStep = #JOB_3_STEP_20) AND "Unit1.Em2.ControlNodes".jrOutPnPLeft.sequence.status.seqActive AND "Unit1.Em2.ControlNodes".jrOutPnPLeft."step".transition1[320],
                         PT := T#100ms);
   IF #statTonTime[320].Q THEN
       "Unit1.Em2.ControlNodes".jrOutPnPLeft.sequence.status.nextStep := #JOB_3_STEP_21;
   END_IF;
END_REGION

REGION Network 27: Step[321] : JR PP Left Clamp Close
   RUNG wire#powerrail
      { S7_Templates := "SrcType := DInt" } EQ_Contact(in1 := "Unit1.Em2.ControlNodes".jrOutPnPLeft.sequence.status.currentStep, in2 := #JOB_3_STEP_21)
      Contact( "Unit1.Em2.ControlNodes".jrOutPnPLeft.sequence.status.seqActive )
      wire#w1
      I_Contact( "Unit1.Em2.ControlNodes".cmJROutPnPLeftClampOpenClose.monitoring.inWorkPos )
      Coil( "Unit1.Em2.ControlNodes".jrOutPnPLeft."step".action1[321] )
   END_RUNG
   RUNG wire#w1
      Contact( "Unit1.Em2.ControlNodes".cmJROutPnPLeftClampOpenClose.monitoring.inWorkPos )
      wire#w2
      { S7_Templates := "SrcType := Variant" } NE_Contact(in1 := #NoDataCheck, in2 := "Unit1.EmData".partData[0])
      wire#w3
      Coil( "Unit1.Em2.ControlNodes".jrOutPnPLeft."step".transition1[321] )
   END_RUNG
   RUNG wire#w2
      I_Contact( "Unit1.Test"."Bool"[40] )
   END_RUNG wire#w3
   RUNG wire#w1
      Contact( "Unit1.Em2.ControlNodes".jrOutPnPLeft."step".transition1[321] )
      { S7_Templates := "time_type := Time" } #statTonTime[321].TON(pt := T#500ms, et =>)
      Move(in := #JOB_3_STEP_22, out1 => "Unit1.Em2.ControlNodes".jrOutPnPLeft.sequence.status.nextStep)
   END_RUNG
   // the same network as SCL:
   #_w1 := ("Unit1.Em2.ControlNodes".jrOutPnPLeft.sequence.status.currentStep = #JOB_3_STEP_21) AND "Unit1.Em2.ControlNodes".jrOutPnPLeft.sequence.status.seqActive;
   "Unit1.Em2.ControlNodes".jrOutPnPLeft."step".action1[321] := #_w1 AND NOT "Unit1.Em2.ControlNodes".cmJROutPnPLeftClampOpenClose.monitoring.inWorkPos;
   "Unit1.Em2.ControlNodes".jrOutPnPLeft."step".transition1[321] := #_w1 AND "Unit1.Em2.ControlNodes".cmJROutPnPLeftClampOpenClose.monitoring.inWorkPos AND ((#NoDataCheck <> "Unit1.EmData".partData[0]) OR NOT "Unit1.Test"."Bool"[40]);
   #statTonTime[321].TON(IN := #_w1 AND "Unit1.Em2.ControlNodes".jrOutPnPLeft."step".transition1[321],
                         PT := T#500ms);
   IF #statTonTime[321].Q THEN
       "Unit1.Em2.ControlNodes".jrOutPnPLeft.sequence.status.nextStep := #JOB_3_STEP_22;
   END_IF;
END_REGION

REGION Network 28: Step[322] : JR PP Left [Request Unclamp] => Stack #2
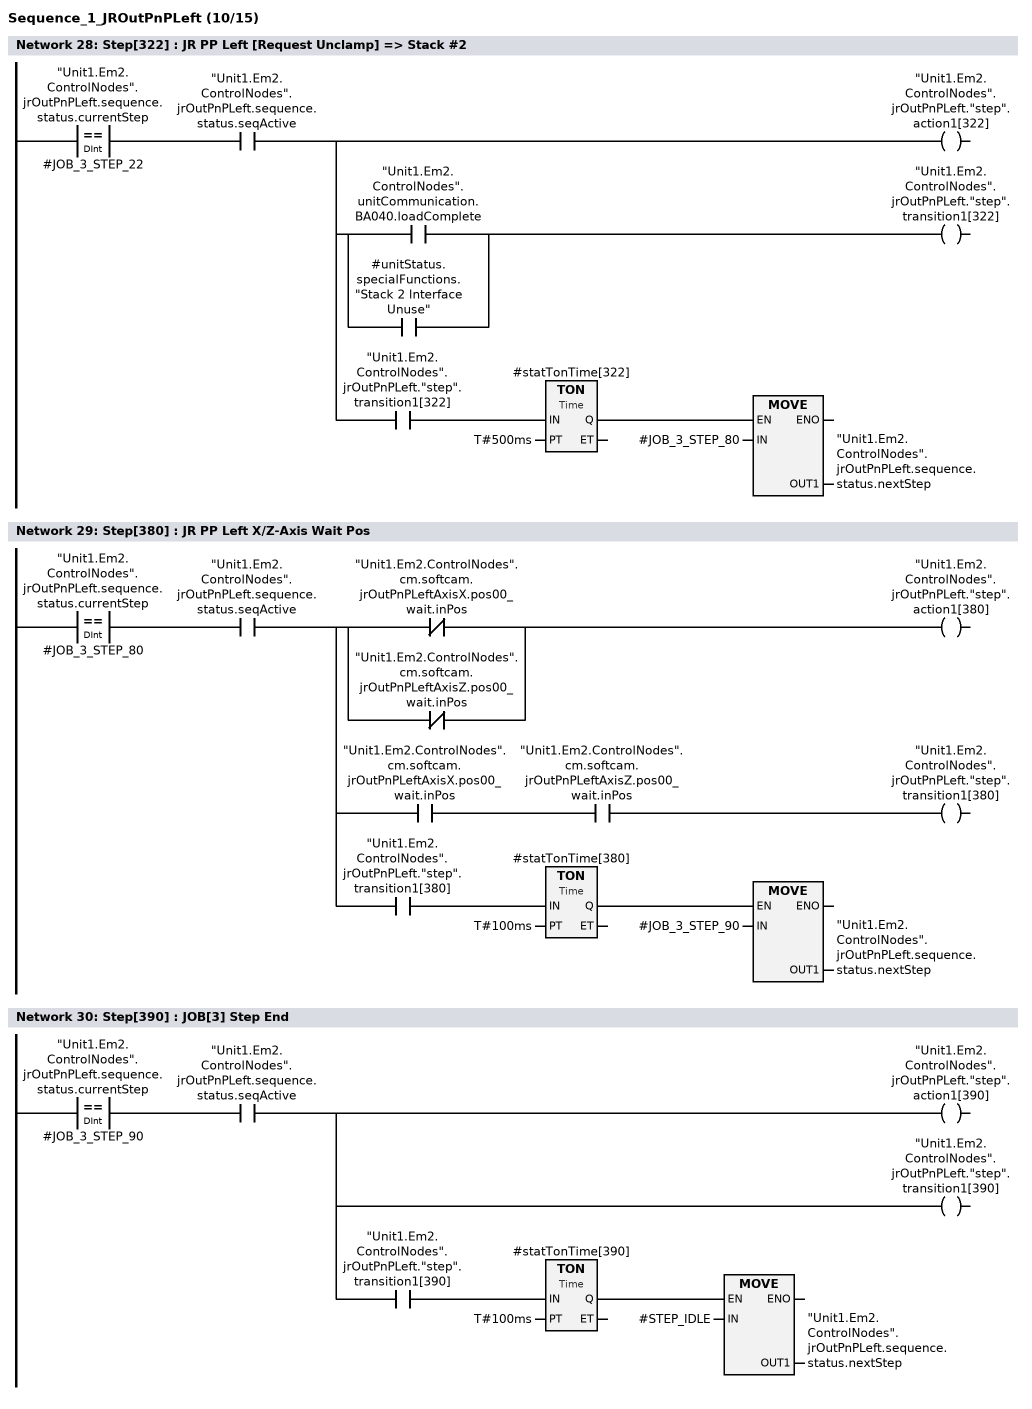
   RUNG wire#powerrail
      { S7_Templates := "SrcType := DInt" } EQ_Contact(in1 := "Unit1.Em2.ControlNodes".jrOutPnPLeft.sequence.status.currentStep, in2 := #JOB_3_STEP_22)
      Contact( "Unit1.Em2.ControlNodes".jrOutPnPLeft.sequence.status.seqActive )
      wire#w1
      Coil( "Unit1.Em2.ControlNodes".jrOutPnPLeft."step".action1[322] )
   END_RUNG
   RUNG wire#w1
      Contact( "Unit1.Em2.ControlNodes".unitCommunication.BA040.loadComplete )
      wire#w2
      Coil( "Unit1.Em2.ControlNodes".jrOutPnPLeft."step".transition1[322] )
   END_RUNG
   RUNG wire#w1
      Contact( #unitStatus.specialFunctions."Stack 2 lnterface Unuse" )
   END_RUNG wire#w2
   RUNG wire#w1
      Contact( "Unit1.Em2.ControlNodes".jrOutPnPLeft."step".transition1[322] )
      { S7_Templates := "time_type := Time" } #statTonTime[322].TON(pt := T#500ms, et =>)
      Move(in := #JOB_3_STEP_80, out1 => "Unit1.Em2.ControlNodes".jrOutPnPLeft.sequence.status.nextStep)
   END_RUNG
   // the same network as SCL:
   "Unit1.Em2.ControlNodes".jrOutPnPLeft."step".action1[322] := ("Unit1.Em2.ControlNodes".jrOutPnPLeft.sequence.status.currentStep = #JOB_3_STEP_22) AND "Unit1.Em2.ControlNodes".jrOutPnPLeft.sequence.status.seqActive;
   "Unit1.Em2.ControlNodes".jrOutPnPLeft."step".transition1[322] := ("Unit1.Em2.ControlNodes".jrOutPnPLeft.sequence.status.currentStep = #JOB_3_STEP_22) AND "Unit1.Em2.ControlNodes".jrOutPnPLeft.sequence.status.seqActive AND ("Unit1.Em2.ControlNodes".unitCommunication.BA040.loadComplete OR #unitStatus.specialFunctions."Stack 2 lnterface Unuse");
   #statTonTime[322].TON(IN := ("Unit1.Em2.ControlNodes".jrOutPnPLeft.sequence.status.currentStep = #JOB_3_STEP_22) AND "Unit1.Em2.ControlNodes".jrOutPnPLeft.sequence.status.seqActive AND "Unit1.Em2.ControlNodes".jrOutPnPLeft."step".transition1[322],
                         PT := T#500ms);
   IF #statTonTime[322].Q THEN
       "Unit1.Em2.ControlNodes".jrOutPnPLeft.sequence.status.nextStep := #JOB_3_STEP_80;
   END_IF;
END_REGION

REGION Network 29: Step[380] : JR PP Left X/Z-Axis Wait Pos
   RUNG wire#powerrail
      { S7_Templates := "SrcType := DInt" } EQ_Contact(in1 := "Unit1.Em2.ControlNodes".jrOutPnPLeft.sequence.status.currentStep, in2 := #JOB_3_STEP_80)
      Contact( "Unit1.Em2.ControlNodes".jrOutPnPLeft.sequence.status.seqActive )
      wire#w1
      I_Contact( "Unit1.Em2.ControlNodes".cm.softcam.jrOutPnPLeftAxisX.pos00_wait.inPos )
      wire#w2
      Coil( "Unit1.Em2.ControlNodes".jrOutPnPLeft."step".action1[380] )
   END_RUNG
   RUNG wire#w1
      I_Contact( "Unit1.Em2.ControlNodes".cm.softcam.jrOutPnPLeftAxisZ.pos00_wait.inPos )
   END_RUNG wire#w2
   RUNG wire#w1
      Contact( "Unit1.Em2.ControlNodes".cm.softcam.jrOutPnPLeftAxisX.pos00_wait.inPos )
      Contact( "Unit1.Em2.ControlNodes".cm.softcam.jrOutPnPLeftAxisZ.pos00_wait.inPos )
      Coil( "Unit1.Em2.ControlNodes".jrOutPnPLeft."step".transition1[380] )
   END_RUNG
   RUNG wire#w1
      Contact( "Unit1.Em2.ControlNodes".jrOutPnPLeft."step".transition1[380] )
      { S7_Templates := "time_type := Time" } #statTonTime[380].TON(pt := T#100ms, et =>)
      Move(in := #JOB_3_STEP_90, out1 => "Unit1.Em2.ControlNodes".jrOutPnPLeft.sequence.status.nextStep)
   END_RUNG
   // the same network as SCL:
   #_w1 := ("Unit1.Em2.ControlNodes".jrOutPnPLeft.sequence.status.currentStep = #JOB_3_STEP_80) AND "Unit1.Em2.ControlNodes".jrOutPnPLeft.sequence.status.seqActive;
   "Unit1.Em2.ControlNodes".jrOutPnPLeft."step".action1[380] := #_w1 AND (NOT "Unit1.Em2.ControlNodes".cm.softcam.jrOutPnPLeftAxisX.pos00_wait.inPos OR NOT "Unit1.Em2.ControlNodes".cm.softcam.jrOutPnPLeftAxisZ.pos00_wait.inPos);
   "Unit1.Em2.ControlNodes".jrOutPnPLeft."step".transition1[380] := #_w1 AND "Unit1.Em2.ControlNodes".cm.softcam.jrOutPnPLeftAxisX.pos00_wait.inPos AND "Unit1.Em2.ControlNodes".cm.softcam.jrOutPnPLeftAxisZ.pos00_wait.inPos;
   #statTonTime[380].TON(IN := #_w1 AND "Unit1.Em2.ControlNodes".jrOutPnPLeft."step".transition1[380],
                         PT := T#100ms);
   IF #statTonTime[380].Q THEN
       "Unit1.Em2.ControlNodes".jrOutPnPLeft.sequence.status.nextStep := #JOB_3_STEP_90;
   END_IF;
END_REGION

REGION Network 30: Step[390] : JOB[3] Step End
   RUNG wire#powerrail
      { S7_Templates := "SrcType := DInt" } EQ_Contact(in1 := "Unit1.Em2.ControlNodes".jrOutPnPLeft.sequence.status.currentStep, in2 := #JOB_3_STEP_90)
      Contact( "Unit1.Em2.ControlNodes".jrOutPnPLeft.sequence.status.seqActive )
      wire#w1
      Coil( "Unit1.Em2.ControlNodes".jrOutPnPLeft."step".action1[390] )
   END_RUNG
   RUNG wire#w1
      Coil( "Unit1.Em2.ControlNodes".jrOutPnPLeft."step".transition1[390] )
   END_RUNG
   RUNG wire#w1
      Contact( "Unit1.Em2.ControlNodes".jrOutPnPLeft."step".transition1[390] )
      { S7_Templates := "time_type := Time" } #statTonTime[390].TON(pt := T#100ms, et =>)
      Move(in := #STEP_IDLE, out1 => "Unit1.Em2.ControlNodes".jrOutPnPLeft.sequence.status.nextStep)
   END_RUNG
   // the same network as SCL:
   "Unit1.Em2.ControlNodes".jrOutPnPLeft."step".action1[390] := ("Unit1.Em2.ControlNodes".jrOutPnPLeft.sequence.status.currentStep = #JOB_3_STEP_90) AND "Unit1.Em2.ControlNodes".jrOutPnPLeft.sequence.status.seqActive;
   "Unit1.Em2.ControlNodes".jrOutPnPLeft."step".transition1[390] := ("Unit1.Em2.ControlNodes".jrOutPnPLeft.sequence.status.currentStep = #JOB_3_STEP_90) AND "Unit1.Em2.ControlNodes".jrOutPnPLeft.sequence.status.seqActive;
   #statTonTime[390].TON(IN := ("Unit1.Em2.ControlNodes".jrOutPnPLeft.sequence.status.currentStep = #JOB_3_STEP_90) AND "Unit1.Em2.ControlNodes".jrOutPnPLeft.sequence.status.seqActive AND "Unit1.Em2.ControlNodes".jrOutPnPLeft."step".transition1[390],
                         PT := T#100ms);
   IF #statTonTime[390].Q THEN
       "Unit1.Em2.ControlNodes".jrOutPnPLeft.sequence.status.nextStep := #STEP_IDLE;
   END_IF;
END_REGION

REGION Network 31: *************** JOB[4] JR PUT TOP TAPE=AUTO *************************
END_REGION

REGION Network 32: Step[401] : JOB[4] Condition
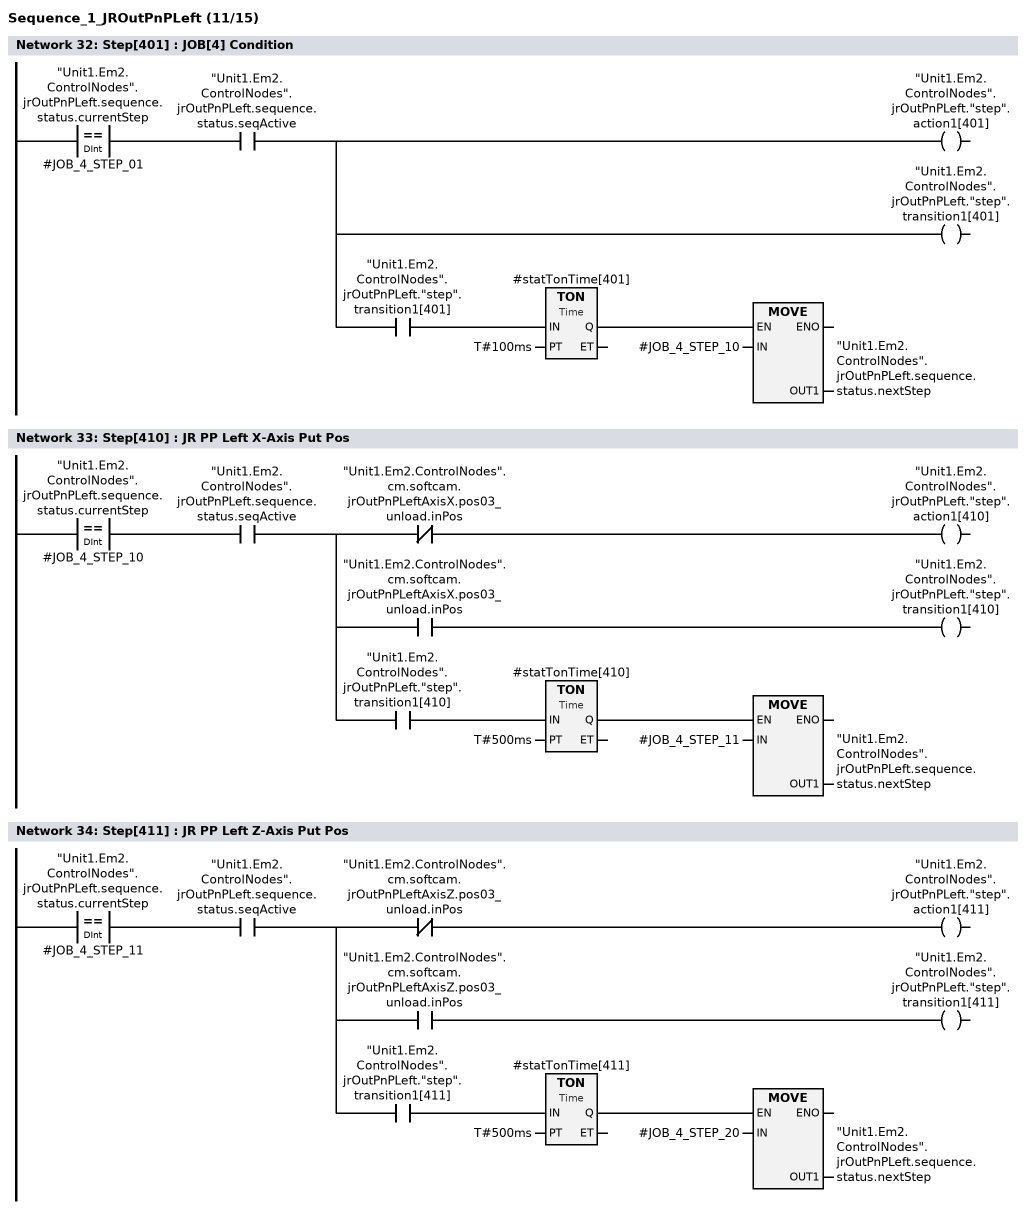
   RUNG wire#powerrail
      { S7_Templates := "SrcType := DInt" } EQ_Contact(in1 := "Unit1.Em2.ControlNodes".jrOutPnPLeft.sequence.status.currentStep, in2 := #JOB_4_STEP_01)
      Contact( "Unit1.Em2.ControlNodes".jrOutPnPLeft.sequence.status.seqActive )
      wire#w1
      Coil( "Unit1.Em2.ControlNodes".jrOutPnPLeft."step".action1[401] )
   END_RUNG
   RUNG wire#w1
      Coil( "Unit1.Em2.ControlNodes".jrOutPnPLeft."step".transition1[401] )
   END_RUNG
   RUNG wire#w1
      Contact( "Unit1.Em2.ControlNodes".jrOutPnPLeft."step".transition1[401] )
      { S7_Templates := "time_type := Time" } #statTonTime[401].TON(pt := T#100ms, et =>)
      Move(in := #JOB_4_STEP_10, out1 => "Unit1.Em2.ControlNodes".jrOutPnPLeft.sequence.status.nextStep)
   END_RUNG
   // the same network as SCL:
   "Unit1.Em2.ControlNodes".jrOutPnPLeft."step".action1[401] := ("Unit1.Em2.ControlNodes".jrOutPnPLeft.sequence.status.currentStep = #JOB_4_STEP_01) AND "Unit1.Em2.ControlNodes".jrOutPnPLeft.sequence.status.seqActive;
   "Unit1.Em2.ControlNodes".jrOutPnPLeft."step".transition1[401] := ("Unit1.Em2.ControlNodes".jrOutPnPLeft.sequence.status.currentStep = #JOB_4_STEP_01) AND "Unit1.Em2.ControlNodes".jrOutPnPLeft.sequence.status.seqActive;
   #statTonTime[401].TON(IN := ("Unit1.Em2.ControlNodes".jrOutPnPLeft.sequence.status.currentStep = #JOB_4_STEP_01) AND "Unit1.Em2.ControlNodes".jrOutPnPLeft.sequence.status.seqActive AND "Unit1.Em2.ControlNodes".jrOutPnPLeft."step".transition1[401],
                         PT := T#100ms);
   IF #statTonTime[401].Q THEN
       "Unit1.Em2.ControlNodes".jrOutPnPLeft.sequence.status.nextStep := #JOB_4_STEP_10;
   END_IF;
END_REGION

REGION Network 33: Step[410] : JR PP Left X-Axis Put Pos
   RUNG wire#powerrail
      { S7_Templates := "SrcType := DInt" } EQ_Contact(in1 := "Unit1.Em2.ControlNodes".jrOutPnPLeft.sequence.status.currentStep, in2 := #JOB_4_STEP_10)
      Contact( "Unit1.Em2.ControlNodes".jrOutPnPLeft.sequence.status.seqActive )
      wire#w1
      I_Contact( "Unit1.Em2.ControlNodes".cm.softcam.jrOutPnPLeftAxisX.pos03_unload.inPos )
      Coil( "Unit1.Em2.ControlNodes".jrOutPnPLeft."step".action1[410] )
   END_RUNG
   RUNG wire#w1
      Contact( "Unit1.Em2.ControlNodes".cm.softcam.jrOutPnPLeftAxisX.pos03_unload.inPos )
      Coil( "Unit1.Em2.ControlNodes".jrOutPnPLeft."step".transition1[410] )
   END_RUNG
   RUNG wire#w1
      Contact( "Unit1.Em2.ControlNodes".jrOutPnPLeft."step".transition1[410] )
      { S7_Templates := "time_type := Time" } #statTonTime[410].TON(pt := T#500ms, et =>)
      Move(in := #JOB_4_STEP_11, out1 => "Unit1.Em2.ControlNodes".jrOutPnPLeft.sequence.status.nextStep)
   END_RUNG
   // the same network as SCL:
   #_w1 := ("Unit1.Em2.ControlNodes".jrOutPnPLeft.sequence.status.currentStep = #JOB_4_STEP_10) AND "Unit1.Em2.ControlNodes".jrOutPnPLeft.sequence.status.seqActive;
   "Unit1.Em2.ControlNodes".jrOutPnPLeft."step".action1[410] := #_w1 AND NOT "Unit1.Em2.ControlNodes".cm.softcam.jrOutPnPLeftAxisX.pos03_unload.inPos;
   "Unit1.Em2.ControlNodes".jrOutPnPLeft."step".transition1[410] := #_w1 AND "Unit1.Em2.ControlNodes".cm.softcam.jrOutPnPLeftAxisX.pos03_unload.inPos;
   #statTonTime[410].TON(IN := #_w1 AND "Unit1.Em2.ControlNodes".jrOutPnPLeft."step".transition1[410],
                         PT := T#500ms);
   IF #statTonTime[410].Q THEN
       "Unit1.Em2.ControlNodes".jrOutPnPLeft.sequence.status.nextStep := #JOB_4_STEP_11;
   END_IF;
END_REGION

REGION Network 34: Step[411] : JR PP Left Z-Axis Put Pos
   RUNG wire#powerrail
      { S7_Templates := "SrcType := DInt" } EQ_Contact(in1 := "Unit1.Em2.ControlNodes".jrOutPnPLeft.sequence.status.currentStep, in2 := #JOB_4_STEP_11)
      Contact( "Unit1.Em2.ControlNodes".jrOutPnPLeft.sequence.status.seqActive )
      wire#w1
      I_Contact( "Unit1.Em2.ControlNodes".cm.softcam.jrOutPnPLeftAxisZ.pos03_unload.inPos )
      Coil( "Unit1.Em2.ControlNodes".jrOutPnPLeft."step".action1[411] )
   END_RUNG
   RUNG wire#w1
      Contact( "Unit1.Em2.ControlNodes".cm.softcam.jrOutPnPLeftAxisZ.pos03_unload.inPos )
      Coil( "Unit1.Em2.ControlNodes".jrOutPnPLeft."step".transition1[411] )
   END_RUNG
   RUNG wire#w1
      Contact( "Unit1.Em2.ControlNodes".jrOutPnPLeft."step".transition1[411] )
      { S7_Templates := "time_type := Time" } #statTonTime[411].TON(pt := T#500ms, et =>)
      Move(in := #JOB_4_STEP_20, out1 => "Unit1.Em2.ControlNodes".jrOutPnPLeft.sequence.status.nextStep)
   END_RUNG
   // the same network as SCL:
   #_w1 := ("Unit1.Em2.ControlNodes".jrOutPnPLeft.sequence.status.currentStep = #JOB_4_STEP_11) AND "Unit1.Em2.ControlNodes".jrOutPnPLeft.sequence.status.seqActive;
   "Unit1.Em2.ControlNodes".jrOutPnPLeft."step".action1[411] := #_w1 AND NOT "Unit1.Em2.ControlNodes".cm.softcam.jrOutPnPLeftAxisZ.pos03_unload.inPos;
   "Unit1.Em2.ControlNodes".jrOutPnPLeft."step".transition1[411] := #_w1 AND "Unit1.Em2.ControlNodes".cm.softcam.jrOutPnPLeftAxisZ.pos03_unload.inPos;
   #statTonTime[411].TON(IN := #_w1 AND "Unit1.Em2.ControlNodes".jrOutPnPLeft."step".transition1[411],
                         PT := T#500ms);
   IF #statTonTime[411].Q THEN
       "Unit1.Em2.ControlNodes".jrOutPnPLeft.sequence.status.nextStep := #JOB_4_STEP_20;
   END_IF;
END_REGION

REGION Network 35: Step[420] : JR PP Left [Unloading Ready] => Top Tape Fix Stage
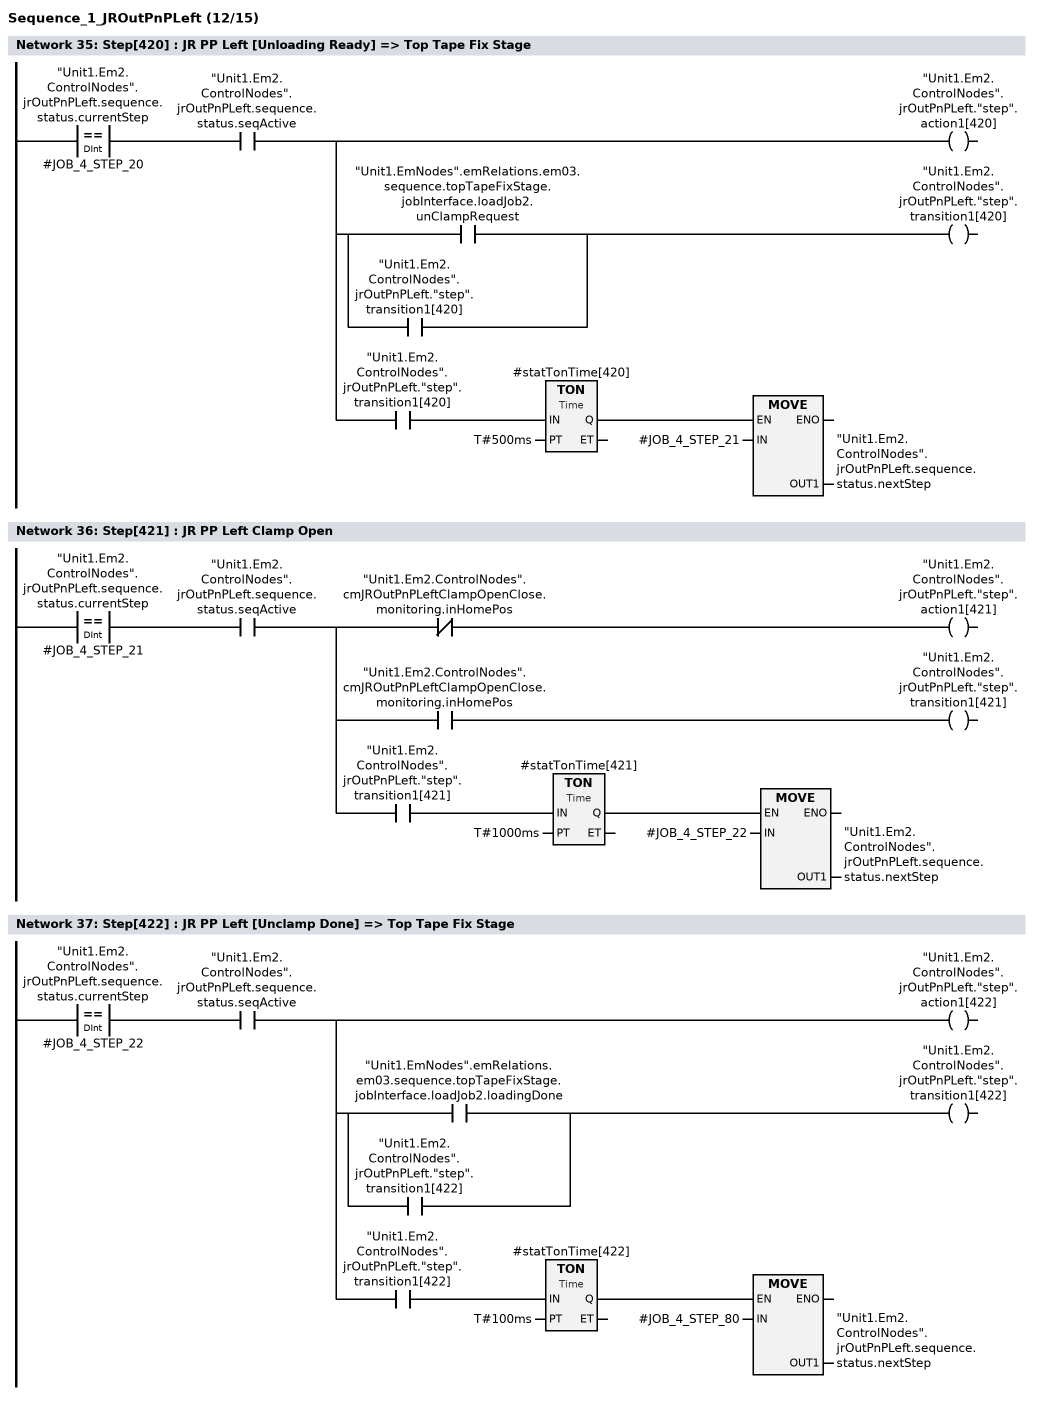
   RUNG wire#powerrail
      { S7_Templates := "SrcType := DInt" } EQ_Contact(in1 := "Unit1.Em2.ControlNodes".jrOutPnPLeft.sequence.status.currentStep, in2 := #JOB_4_STEP_20)
      Contact( "Unit1.Em2.ControlNodes".jrOutPnPLeft.sequence.status.seqActive )
      wire#w1
      Coil( "Unit1.Em2.ControlNodes".jrOutPnPLeft."step".action1[420] )
   END_RUNG
   RUNG wire#w1
      Contact( "Unit1.EmNodes".emRelations.em03.sequence.topTapeFixStage.jobInterface.loadJob2.unClampRequest )
      wire#w2
      Coil( "Unit1.Em2.ControlNodes".jrOutPnPLeft."step".transition1[420] )
   END_RUNG
   RUNG wire#w1
      Contact( "Unit1.Em2.ControlNodes".jrOutPnPLeft."step".transition1[420] )
   END_RUNG wire#w2
   RUNG wire#w1
      Contact( "Unit1.Em2.ControlNodes".jrOutPnPLeft."step".transition1[420] )
      { S7_Templates := "time_type := Time" } #statTonTime[420].TON(pt := T#500ms, et =>)
      Move(in := #JOB_4_STEP_21, out1 => "Unit1.Em2.ControlNodes".jrOutPnPLeft.sequence.status.nextStep)
   END_RUNG
   // the same network as SCL:
   "Unit1.Em2.ControlNodes".jrOutPnPLeft."step".action1[420] := ("Unit1.Em2.ControlNodes".jrOutPnPLeft.sequence.status.currentStep = #JOB_4_STEP_20) AND "Unit1.Em2.ControlNodes".jrOutPnPLeft.sequence.status.seqActive;
   "Unit1.Em2.ControlNodes".jrOutPnPLeft."step".transition1[420] := ("Unit1.Em2.ControlNodes".jrOutPnPLeft.sequence.status.currentStep = #JOB_4_STEP_20) AND "Unit1.Em2.ControlNodes".jrOutPnPLeft.sequence.status.seqActive AND ("Unit1.EmNodes".emRelations.em03.sequence.topTapeFixStage.jobInterface.loadJob2.unClampRequest OR "Unit1.Em2.ControlNodes".jrOutPnPLeft."step".transition1[420]);
   #statTonTime[420].TON(IN := ("Unit1.Em2.ControlNodes".jrOutPnPLeft.sequence.status.currentStep = #JOB_4_STEP_20) AND "Unit1.Em2.ControlNodes".jrOutPnPLeft.sequence.status.seqActive AND "Unit1.Em2.ControlNodes".jrOutPnPLeft."step".transition1[420],
                         PT := T#500ms);
   IF #statTonTime[420].Q THEN
       "Unit1.Em2.ControlNodes".jrOutPnPLeft.sequence.status.nextStep := #JOB_4_STEP_21;
   END_IF;
END_REGION

REGION Network 36: Step[421] : JR PP Left Clamp Open
   RUNG wire#powerrail
      { S7_Templates := "SrcType := DInt" } EQ_Contact(in1 := "Unit1.Em2.ControlNodes".jrOutPnPLeft.sequence.status.currentStep, in2 := #JOB_4_STEP_21)
      Contact( "Unit1.Em2.ControlNodes".jrOutPnPLeft.sequence.status.seqActive )
      wire#w1
      I_Contact( "Unit1.Em2.ControlNodes".cmJROutPnPLeftClampOpenClose.monitoring.inHomePos )
      Coil( "Unit1.Em2.ControlNodes".jrOutPnPLeft."step".action1[421] )
   END_RUNG
   RUNG wire#w1
      Contact( "Unit1.Em2.ControlNodes".cmJROutPnPLeftClampOpenClose.monitoring.inHomePos )
      Coil( "Unit1.Em2.ControlNodes".jrOutPnPLeft."step".transition1[421] )
   END_RUNG
   RUNG wire#w1
      Contact( "Unit1.Em2.ControlNodes".jrOutPnPLeft."step".transition1[421] )
      { S7_Templates := "time_type := Time" } #statTonTime[421].TON(pt := T#1000ms, et =>)
      Move(in := #JOB_4_STEP_22, out1 => "Unit1.Em2.ControlNodes".jrOutPnPLeft.sequence.status.nextStep)
   END_RUNG
   // the same network as SCL:
   #_w1 := ("Unit1.Em2.ControlNodes".jrOutPnPLeft.sequence.status.currentStep = #JOB_4_STEP_21) AND "Unit1.Em2.ControlNodes".jrOutPnPLeft.sequence.status.seqActive;
   "Unit1.Em2.ControlNodes".jrOutPnPLeft."step".action1[421] := #_w1 AND NOT "Unit1.Em2.ControlNodes".cmJROutPnPLeftClampOpenClose.monitoring.inHomePos;
   "Unit1.Em2.ControlNodes".jrOutPnPLeft."step".transition1[421] := #_w1 AND "Unit1.Em2.ControlNodes".cmJROutPnPLeftClampOpenClose.monitoring.inHomePos;
   #statTonTime[421].TON(IN := #_w1 AND "Unit1.Em2.ControlNodes".jrOutPnPLeft."step".transition1[421],
                         PT := T#1000ms);
   IF #statTonTime[421].Q THEN
       "Unit1.Em2.ControlNodes".jrOutPnPLeft.sequence.status.nextStep := #JOB_4_STEP_22;
   END_IF;
END_REGION

REGION Network 37: Step[422] : JR PP Left [Unclamp Done] => Top Tape Fix Stage
   RUNG wire#powerrail
      { S7_Templates := "SrcType := DInt" } EQ_Contact(in1 := "Unit1.Em2.ControlNodes".jrOutPnPLeft.sequence.status.currentStep, in2 := #JOB_4_STEP_22)
      Contact( "Unit1.Em2.ControlNodes".jrOutPnPLeft.sequence.status.seqActive )
      wire#w1
      Coil( "Unit1.Em2.ControlNodes".jrOutPnPLeft."step".action1[422] )
   END_RUNG
   RUNG wire#w1
      Contact( "Unit1.EmNodes".emRelations.em03.sequence.topTapeFixStage.jobInterface.loadJob2.loadingDone )
      wire#w2
      Coil( "Unit1.Em2.ControlNodes".jrOutPnPLeft."step".transition1[422] )
   END_RUNG
   RUNG wire#w1
      Contact( "Unit1.Em2.ControlNodes".jrOutPnPLeft."step".transition1[422] )
   END_RUNG wire#w2
   RUNG wire#w1
      Contact( "Unit1.Em2.ControlNodes".jrOutPnPLeft."step".transition1[422] )
      { S7_Templates := "time_type := Time" } #statTonTime[422].TON(pt := T#100ms, et =>)
      Move(in := #JOB_4_STEP_80, out1 => "Unit1.Em2.ControlNodes".jrOutPnPLeft.sequence.status.nextStep)
   END_RUNG
   // the same network as SCL:
   "Unit1.Em2.ControlNodes".jrOutPnPLeft."step".action1[422] := ("Unit1.Em2.ControlNodes".jrOutPnPLeft.sequence.status.currentStep = #JOB_4_STEP_22) AND "Unit1.Em2.ControlNodes".jrOutPnPLeft.sequence.status.seqActive;
   "Unit1.Em2.ControlNodes".jrOutPnPLeft."step".transition1[422] := ("Unit1.Em2.ControlNodes".jrOutPnPLeft.sequence.status.currentStep = #JOB_4_STEP_22) AND "Unit1.Em2.ControlNodes".jrOutPnPLeft.sequence.status.seqActive AND ("Unit1.EmNodes".emRelations.em03.sequence.topTapeFixStage.jobInterface.loadJob2.loadingDone OR "Unit1.Em2.ControlNodes".jrOutPnPLeft."step".transition1[422]);
   #statTonTime[422].TON(IN := ("Unit1.Em2.ControlNodes".jrOutPnPLeft.sequence.status.currentStep = #JOB_4_STEP_22) AND "Unit1.Em2.ControlNodes".jrOutPnPLeft.sequence.status.seqActive AND "Unit1.Em2.ControlNodes".jrOutPnPLeft."step".transition1[422],
                         PT := T#100ms);
   IF #statTonTime[422].Q THEN
       "Unit1.Em2.ControlNodes".jrOutPnPLeft.sequence.status.nextStep := #JOB_4_STEP_80;
   END_IF;
END_REGION

REGION Network 38: Step[480] : JR PP Left X/Z-Axis Wait Pos
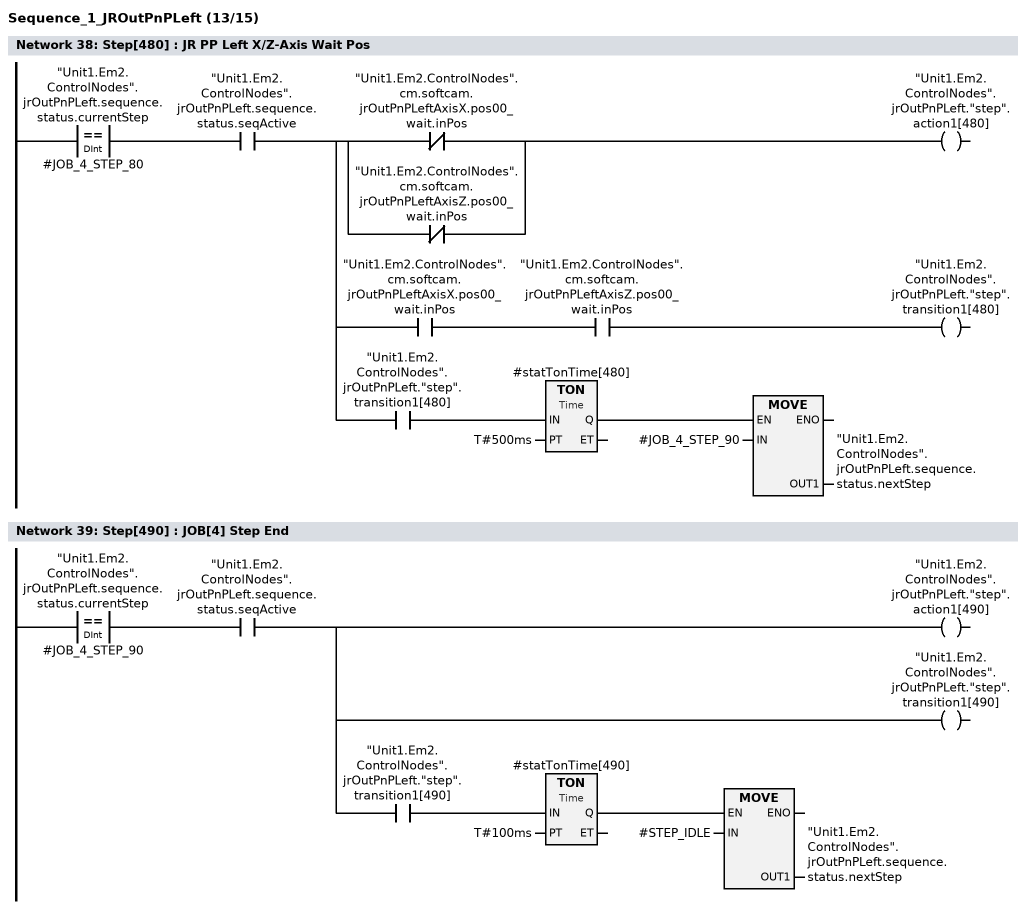
   RUNG wire#powerrail
      { S7_Templates := "SrcType := DInt" } EQ_Contact(in1 := "Unit1.Em2.ControlNodes".jrOutPnPLeft.sequence.status.currentStep, in2 := #JOB_4_STEP_80)
      Contact( "Unit1.Em2.ControlNodes".jrOutPnPLeft.sequence.status.seqActive )
      wire#w1
      I_Contact( "Unit1.Em2.ControlNodes".cm.softcam.jrOutPnPLeftAxisX.pos00_wait.inPos )
      wire#w2
      Coil( "Unit1.Em2.ControlNodes".jrOutPnPLeft."step".action1[480] )
   END_RUNG
   RUNG wire#w1
      I_Contact( "Unit1.Em2.ControlNodes".cm.softcam.jrOutPnPLeftAxisZ.pos00_wait.inPos )
   END_RUNG wire#w2
   RUNG wire#w1
      Contact( "Unit1.Em2.ControlNodes".cm.softcam.jrOutPnPLeftAxisX.pos00_wait.inPos )
      Contact( "Unit1.Em2.ControlNodes".cm.softcam.jrOutPnPLeftAxisZ.pos00_wait.inPos )
      Coil( "Unit1.Em2.ControlNodes".jrOutPnPLeft."step".transition1[480] )
   END_RUNG
   RUNG wire#w1
      Contact( "Unit1.Em2.ControlNodes".jrOutPnPLeft."step".transition1[480] )
      { S7_Templates := "time_type := Time" } #statTonTime[480].TON(pt := T#500ms, et =>)
      Move(in := #JOB_4_STEP_90, out1 => "Unit1.Em2.ControlNodes".jrOutPnPLeft.sequence.status.nextStep)
   END_RUNG
   // the same network as SCL:
   #_w1 := ("Unit1.Em2.ControlNodes".jrOutPnPLeft.sequence.status.currentStep = #JOB_4_STEP_80) AND "Unit1.Em2.ControlNodes".jrOutPnPLeft.sequence.status.seqActive;
   "Unit1.Em2.ControlNodes".jrOutPnPLeft."step".action1[480] := #_w1 AND (NOT "Unit1.Em2.ControlNodes".cm.softcam.jrOutPnPLeftAxisX.pos00_wait.inPos OR NOT "Unit1.Em2.ControlNodes".cm.softcam.jrOutPnPLeftAxisZ.pos00_wait.inPos);
   "Unit1.Em2.ControlNodes".jrOutPnPLeft."step".transition1[480] := #_w1 AND "Unit1.Em2.ControlNodes".cm.softcam.jrOutPnPLeftAxisX.pos00_wait.inPos AND "Unit1.Em2.ControlNodes".cm.softcam.jrOutPnPLeftAxisZ.pos00_wait.inPos;
   #statTonTime[480].TON(IN := #_w1 AND "Unit1.Em2.ControlNodes".jrOutPnPLeft."step".transition1[480],
                         PT := T#500ms);
   IF #statTonTime[480].Q THEN
       "Unit1.Em2.ControlNodes".jrOutPnPLeft.sequence.status.nextStep := #JOB_4_STEP_90;
   END_IF;
END_REGION

REGION Network 39: Step[490] : JOB[4] Step End
   RUNG wire#powerrail
      { S7_Templates := "SrcType := DInt" } EQ_Contact(in1 := "Unit1.Em2.ControlNodes".jrOutPnPLeft.sequence.status.currentStep, in2 := #JOB_4_STEP_90)
      Contact( "Unit1.Em2.ControlNodes".jrOutPnPLeft.sequence.status.seqActive )
      wire#w1
      Coil( "Unit1.Em2.ControlNodes".jrOutPnPLeft."step".action1[490] )
   END_RUNG
   RUNG wire#w1
      Coil( "Unit1.Em2.ControlNodes".jrOutPnPLeft."step".transition1[490] )
   END_RUNG
   RUNG wire#w1
      Contact( "Unit1.Em2.ControlNodes".jrOutPnPLeft."step".transition1[490] )
      { S7_Templates := "time_type := Time" } #statTonTime[490].TON(pt := T#100ms, et =>)
      Move(in := #STEP_IDLE, out1 => "Unit1.Em2.ControlNodes".jrOutPnPLeft.sequence.status.nextStep)
   END_RUNG
   // the same network as SCL:
   "Unit1.Em2.ControlNodes".jrOutPnPLeft."step".action1[490] := ("Unit1.Em2.ControlNodes".jrOutPnPLeft.sequence.status.currentStep = #JOB_4_STEP_90) AND "Unit1.Em2.ControlNodes".jrOutPnPLeft.sequence.status.seqActive;
   "Unit1.Em2.ControlNodes".jrOutPnPLeft."step".transition1[490] := ("Unit1.Em2.ControlNodes".jrOutPnPLeft.sequence.status.currentStep = #JOB_4_STEP_90) AND "Unit1.Em2.ControlNodes".jrOutPnPLeft.sequence.status.seqActive;
   #statTonTime[490].TON(IN := ("Unit1.Em2.ControlNodes".jrOutPnPLeft.sequence.status.currentStep = #JOB_4_STEP_90) AND "Unit1.Em2.ControlNodes".jrOutPnPLeft.sequence.status.seqActive AND "Unit1.Em2.ControlNodes".jrOutPnPLeft."step".transition1[490],
                         PT := T#100ms);
   IF #statTonTime[490].Q THEN
       "Unit1.Em2.ControlNodes".jrOutPnPLeft.sequence.status.nextStep := #STEP_IDLE;
   END_IF;
END_REGION

REGION Network 40: *************** IMMEDIATE STOP ****************
END_REGION

REGION Network 41: Immediate Stop
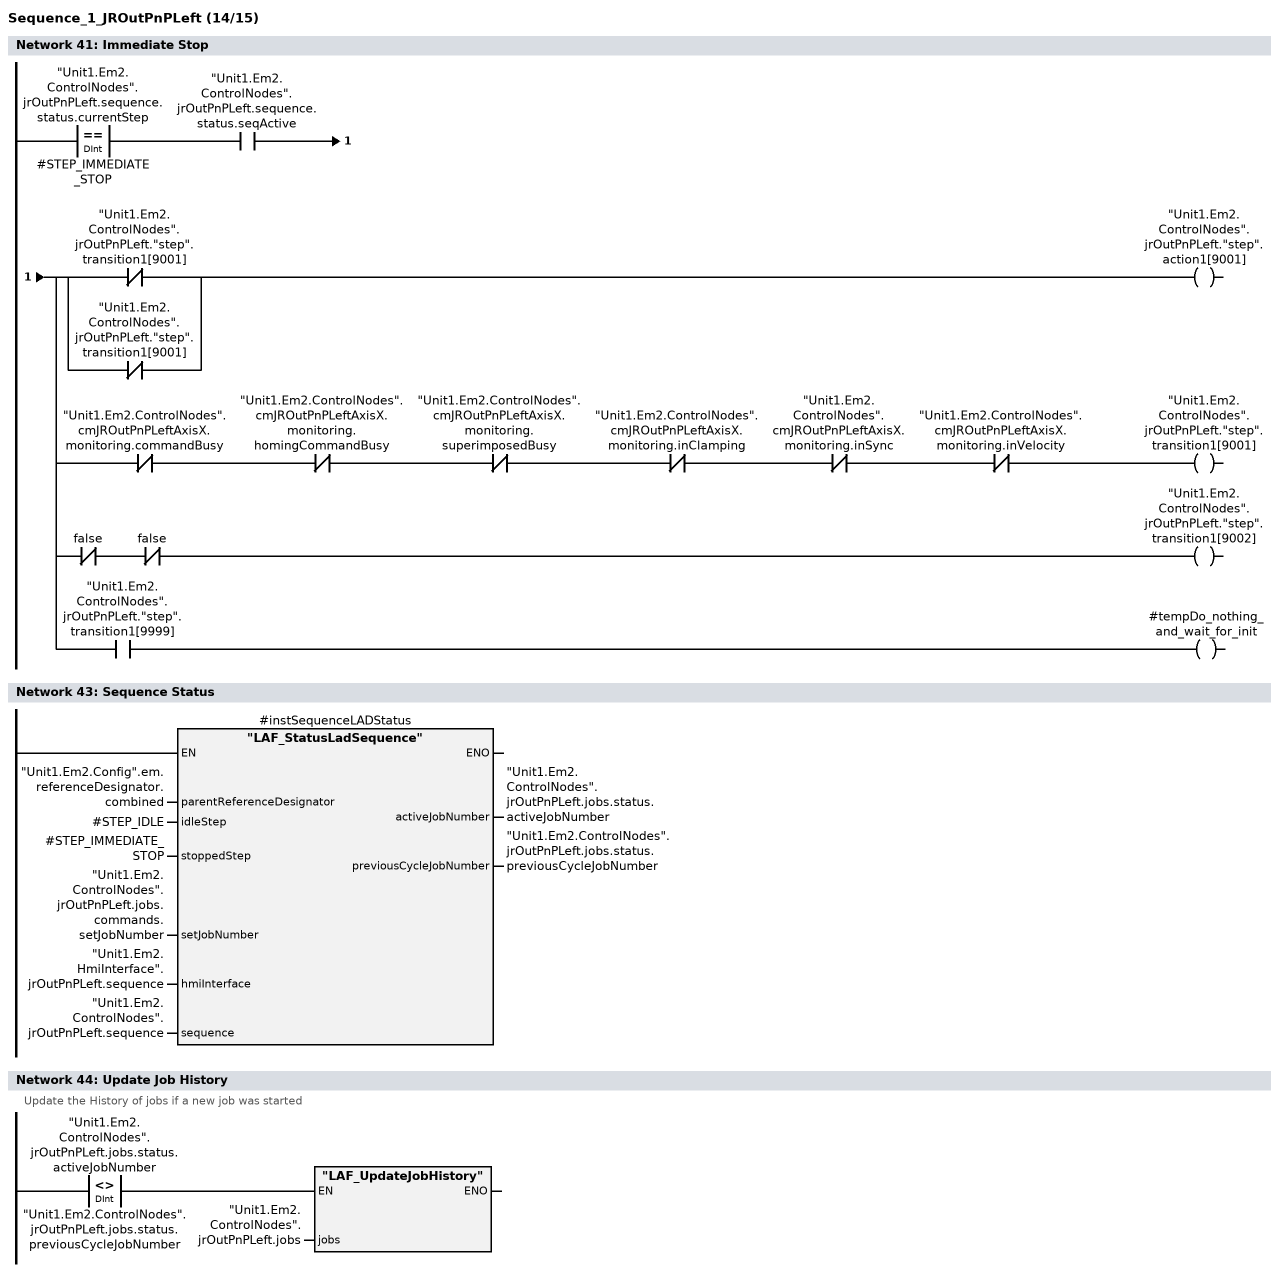
   RUNG wire#powerrail
      { S7_Templates := "SrcType := DInt" } EQ_Contact(in1 := "Unit1.Em2.ControlNodes".jrOutPnPLeft.sequence.status.currentStep, in2 := #STEP_IMMEDIATE_STOP)
      Contact( "Unit1.Em2.ControlNodes".jrOutPnPLeft.sequence.status.seqActive )
      wire#w1
      I_Contact( "Unit1.Em2.ControlNodes".jrOutPnPLeft."step".transition1[9001] )
      wire#w2
      Coil( "Unit1.Em2.ControlNodes".jrOutPnPLeft."step".action1[9001] )
   END_RUNG
   RUNG wire#w1
      I_Contact( "Unit1.Em2.ControlNodes".jrOutPnPLeft."step".transition1[9001] )
   END_RUNG wire#w2
   RUNG wire#w1
      I_Contact( "Unit1.Em2.ControlNodes".cmJROutPnPLeftAxisX.monitoring.commandBusy )
      I_Contact( "Unit1.Em2.ControlNodes".cmJROutPnPLeftAxisX.monitoring.homingCommandBusy )
      I_Contact( "Unit1.Em2.ControlNodes".cmJROutPnPLeftAxisX.monitoring.superimposedBusy )
      I_Contact( "Unit1.Em2.ControlNodes".cmJROutPnPLeftAxisX.monitoring.inClamping )
      I_Contact( "Unit1.Em2.ControlNodes".cmJROutPnPLeftAxisX.monitoring.inSync )
      I_Contact( "Unit1.Em2.ControlNodes".cmJROutPnPLeftAxisX.monitoring.inVelocity )
      Coil( "Unit1.Em2.ControlNodes".jrOutPnPLeft."step".transition1[9001] )
   END_RUNG
   RUNG wire#w1
      I_Contact( false )
      I_Contact( false )
      Coil( "Unit1.Em2.ControlNodes".jrOutPnPLeft."step".transition1[9002] )
   END_RUNG
   RUNG wire#w1
      Contact( "Unit1.Em2.ControlNodes".jrOutPnPLeft."step".transition1[9999] )
      Coil( #tempDo_nothing_and_wait_for_init )
   END_RUNG
   // the same network as SCL:
   #_w1 := ("Unit1.Em2.ControlNodes".jrOutPnPLeft.sequence.status.currentStep = #STEP_IMMEDIATE_STOP) AND "Unit1.Em2.ControlNodes".jrOutPnPLeft.sequence.status.seqActive;
   "Unit1.Em2.ControlNodes".jrOutPnPLeft."step".action1[9001] := #_w1 AND (NOT "Unit1.Em2.ControlNodes".jrOutPnPLeft."step".transition1[9001] OR NOT "Unit1.Em2.ControlNodes".jrOutPnPLeft."step".transition1[9001]);
   "Unit1.Em2.ControlNodes".jrOutPnPLeft."step".transition1[9001] := #_w1 AND NOT "Unit1.Em2.ControlNodes".cmJROutPnPLeftAxisX.monitoring.commandBusy AND NOT "Unit1.Em2.ControlNodes".cmJROutPnPLeftAxisX.monitoring.homingCommandBusy AND NOT "Unit1.Em2.ControlNodes".cmJROutPnPLeftAxisX.monitoring.superimposedBusy AND NOT "Unit1.Em2.ControlNodes".cmJROutPnPLeftAxisX.monitoring.inClamping AND NOT "Unit1.Em2.ControlNodes".cmJROutPnPLeftAxisX.monitoring.inSync AND NOT "Unit1.Em2.ControlNodes".cmJROutPnPLeftAxisX.monitoring.inVelocity;
   "Unit1.Em2.ControlNodes".jrOutPnPLeft."step".transition1[9002] := #_w1 AND NOT false AND NOT false;
   #tempDo_nothing_and_wait_for_init := #_w1 AND "Unit1.Em2.ControlNodes".jrOutPnPLeft."step".transition1[9999];
END_REGION

REGION Network 42: *************** STATUS **********************
END_REGION

REGION Network 43: Sequence Status
   RUNG wire#powerrail
      #instSequenceLADStatus(parentReferenceDesignator := "Unit1.Em2.Config".em.referenceDesignator.combined, idleStep := #STEP_IDLE, stoppedStep := #STEP_IMMEDIATE_STOP, setJobNumber := "Unit1.Em2.ControlNodes".jrOutPnPLeft.jobs.commands.setJobNumber, hmiInterface := "Unit1.Em2.HmiInterface".jrOutPnPLeft.sequence, sequence := "Unit1.Em2.ControlNodes".jrOutPnPLeft.sequence, activeJobNumber => "Unit1.Em2.ControlNodes".jrOutPnPLeft.jobs.status.activeJobNumber, previousCycleJobNumber => "Unit1.Em2.ControlNodes".jrOutPnPLeft.jobs.status.previousCycleJobNumber)
   END_RUNG
   // the same network as SCL:
   #instSequenceLADStatus(parentReferenceDesignator := "Unit1.Em2.Config".em.referenceDesignator.combined,   // "LAF_StatusLadSequence"
                          idleStep := #STEP_IDLE,
                          stoppedStep := #STEP_IMMEDIATE_STOP,
                          setJobNumber := "Unit1.Em2.ControlNodes".jrOutPnPLeft.jobs.commands.setJobNumber,
                          hmiInterface := "Unit1.Em2.HmiInterface".jrOutPnPLeft.sequence,
                          sequence := "Unit1.Em2.ControlNodes".jrOutPnPLeft.sequence,
                          activeJobNumber => "Unit1.Em2.ControlNodes".jrOutPnPLeft.jobs.status.activeJobNumber,
                          previousCycleJobNumber => "Unit1.Em2.ControlNodes".jrOutPnPLeft.jobs.status.previousCycleJobNumber);
END_REGION

REGION Network 44: Update Job History
   // Update the History of jobs if a new job was started
   RUNG wire#powerrail
      { S7_Templates := "SrcType := DInt" } NE_Contact(in1 := "Unit1.Em2.ControlNodes".jrOutPnPLeft.jobs.status.activeJobNumber, in2 := "Unit1.Em2.ControlNodes".jrOutPnPLeft.jobs.status.previousCycleJobNumber)
      "LAF_UpdateJobHistory"(jobs := "Unit1.Em2.ControlNodes".jrOutPnPLeft.jobs)
   END_RUNG
   // the same network as SCL:
   IF "Unit1.Em2.ControlNodes".jrOutPnPLeft.jobs.status.activeJobNumber <> "Unit1.Em2.ControlNodes".jrOutPnPLeft.jobs.status.previousCycleJobNumber THEN
       "LAF_UpdateJobHistory"(jobs := "Unit1.Em2.ControlNodes".jrOutPnPLeft.jobs);
   END_IF;
END_REGION

REGION Network 45: Output steps as String
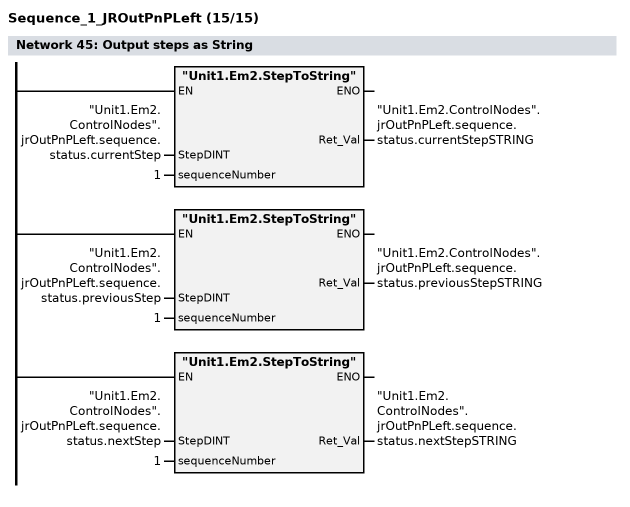
   RUNG wire#powerrail
      "Unit1.Em2.StepToString"(StepDINT := "Unit1.Em2.ControlNodes".jrOutPnPLeft.sequence.status.currentStep, sequenceNumber := 1, Ret_Val => "Unit1.Em2.ControlNodes".jrOutPnPLeft.sequence.status.currentStepSTRING)
   END_RUNG
   RUNG wire#powerrail
      "Unit1.Em2.StepToString"(StepDINT := "Unit1.Em2.ControlNodes".jrOutPnPLeft.sequence.status.previousStep, sequenceNumber := 1, Ret_Val => "Unit1.Em2.ControlNodes".jrOutPnPLeft.sequence.status.previousStepSTRING)
   END_RUNG
   RUNG wire#powerrail
      "Unit1.Em2.StepToString"(StepDINT := "Unit1.Em2.ControlNodes".jrOutPnPLeft.sequence.status.nextStep, sequenceNumber := 1, Ret_Val => "Unit1.Em2.ControlNodes".jrOutPnPLeft.sequence.status.nextStepSTRING)
   END_RUNG
   // the same network as SCL:
   "Unit1.Em2.ControlNodes".jrOutPnPLeft.sequence.status.currentStepSTRING := "Unit1.Em2.StepToString"(StepDINT := "Unit1.Em2.ControlNodes".jrOutPnPLeft.sequence.status.currentStep,
                           sequenceNumber := 1);
   "Unit1.Em2.ControlNodes".jrOutPnPLeft.sequence.status.previousStepSTRING := "Unit1.Em2.StepToString"(StepDINT := "Unit1.Em2.ControlNodes".jrOutPnPLeft.sequence.status.previousStep,
                           sequenceNumber := 1);
   "Unit1.Em2.ControlNodes".jrOutPnPLeft.sequence.status.nextStepSTRING := "Unit1.Em2.StepToString"(StepDINT := "Unit1.Em2.ControlNodes".jrOutPnPLeft.sequence.status.nextStep,
                           sequenceNumber := 1);
END_REGION
END_FUNCTION_BLOCK
